// TIA Portal project "1_TIA" (V17)

(* hardware
DEVICE "S7-1200 station_1"  S7-1200 Station
   slot 0: "Rack_0"  S7-1200 Rack  Rack  V1.0
   slot 1: "STATION_1"  CPU 1215C DC/DC/DC  6ES7 215-1AG40-0XB0  V4.4
DEVICE "S7-1200 station_2"  S7-1200 Station
   slot 0: "Rack_0"  S7-1200 Rack  Rack  V1.0
   slot 1: "STATION_2"  CPU 1215C DC/DC/DC  6ES7 215-1AG40-0XB0  V4.4
*)

// ===== PLC "STATION_1"  CPU 1215C DC/DC/DC =====

VAR_GLOBAL   // PLC tag table "Default tag table"
   "Clock_Byte" AT %MB0 : Byte;
   "Clock_10Hz" AT %M0.0 : Bool;
   "Clock_5Hz" AT %M0.1 : Bool;
   "Clock_2.5Hz" AT %M0.2 : Bool;
   "Clock_2Hz" AT %M0.3 : Bool;
   "Clock_1.25Hz" AT %M0.4 : Bool;
   "Clock_1Hz" AT %M0.5 : Bool;
   "Clock_0.625Hz" AT %M0.6 : Bool;
   "Clock_0.5Hz" AT %M0.7 : Bool;
   "System_Byte" AT %MB1 : Byte;
   "FirstScan" AT %M1.0 : Bool;
   "DiagStatusUpdate" AT %M1.1 : Bool;
   "AlwaysTRUE" AT %M1.2 : Bool;
   "AlwaysFALSE" AT %M1.3 : Bool;
   "XUNG_PTRIG_1" AT %M10.0 : Bool;
   "XUNG_PTRIG_2" AT %M10.1 : Bool;
   "XUNG_PTRIG_3" AT %M10.2 : Bool;
   "XUNG_PTRIG_4" AT %M10.3 : Bool;
   "XUNG_PTRIG_5" AT %M10.4 : Bool;
   "XUNG_PTRIG_6" AT %M10.5 : Bool;
   "XUNG_PTRIG_7" AT %M10.6 : Bool;
   "XUNG_PTRIG_8" AT %M10.7 : Bool;
END_VAR

VAR_GLOBAL   // PLC tag table "Input"
   "Fault_Valve_1" AT %I0.0 : Bool;   // Bit báo lỗi van 1
   "Fault_Valve_2" AT %I0.1 : Bool;   // Bit báo lỗi van 2
   "Fault_Valve_3" AT %I0.2 : Bool;   // Bit báo lỗi van 3
   "FAULT_DC_TRON" AT %I0.3 : Bool;   // Bit báo lỗi động cơ trộn
   "Auto" AT %I0.5 : Bool;   // Chế độ Auto
   "Manual" AT %I0.6 : Bool;   // Chế độ Manual
   "FAULT_DC_EXPORT" AT %I0.4 : Bool;   // Bit baso lỗi máy đóng gói
   "ON" AT %I0.7 : Bool;   // Bật Hệ thống
   "OFF" AT %I1.0 : Bool;   // Tắt hệ thống
END_VAR

VAR_GLOBAL   // PLC tag table "Output"
   "Q_VALVE_1" AT %Q0.0 : Bool;   // Đầu ra van 1
   "Q_VALVE_2" AT %Q0.1 : Bool;   // Đầu ra van 2
   "Q_VALVE_3" AT %Q0.2 : Bool;   // Đầu ra van 3
   "Q_DC_TRON" AT %Q0.3 : Bool;   // Đầu ra động cơ trộn
   "Q_Lamp_Auto" AT %Q0.5 : Bool;
   "Q_Lamp_Manu" AT %Q0.6 : Bool;
   "Q_DC_Export" AT %Q0.4 : Bool;   // Đầu ra máy đóng gói
   "Q_System" AT %Q0.7 : Bool;
END_VAR

VAR_GLOBAL   // PLC tag table "simulation"
   "Simu_Fault_Valve_1" AT %M20.0 : Bool;
   "Simu_Fault_Valve_2" AT %M20.1 : Bool;
   "Simu_Fault_Valve_3" AT %M20.2 : Bool;
   "Simu_Fault_DC_TRON" AT %M20.3 : Bool;
   "Simu_Fault_DC_EXPORT" AT %M20.4 : Bool;
END_VAR

DATA_BLOCK "DB_Webserver"   // DB1
{ S7_Optimized_Access := 'FALSE' }
VERSION : 0.1
   VAR
      btt_Auto : Bool;   // Nút nhấn chế độ tự động
      btt_Manu : Bool;   // Nút nhấn chế độ bằng tay
      btt_Auto_Confirm : Bool;   // Nút nhấn xác nhận
      btt_V1_Open : Bool;   // Nút nhấn chế độ bằng tay mở van 1
      btt_V1_Close : Bool;   // Nút nhấn chế độ bằng tay đóng van 1
      btt_V2_Open : Bool;   // Nút nhấn chế độ bằng tay mở van 2
      btt_V2_Close : Bool;   // Nút nhấn chế độ bằng tay đóng van 2
      btt_V3_Open : Bool;   // Nút nhấn chế độ bằng tay mở van 3
      btt_V3_Close : Bool;   // Nút nhấn chế độ bằng tay đóng van 3
      btt_DC_Tron_Run : Bool;   // Nút nhấn chế độ bằng tay chạy ĐC trộn
      btt_DC_Tron_Stop : Bool;   // Nút nhấn chế độ bằng tay dừng ĐC trộn
      btt_DC_Export_Run : Bool;   // Nút nhấn chế độ bằng tay chạy máy đóng gói
      btt_DC_Export_Stop : Bool;   // Nút nhấn chế độ bằng tay đóng máy đóng gói
      CB_Can : Bool;   // Cảm biến cạn bồn trộn
      Q_Lamp_Auto : Bool;   // Đèn chế độ tự động
      Q_Lamp_Manu : Bool;   // Đèn chế độ bằng tay
      status_Valve_1 : Byte;   // Trạng thái van 1 (0 = Đang đóng, 1 = Đang mở, 2 = Đang lỗi)
      status_Valve_2 : Byte;   // Trạng thái van 2 (0 = Đang đóng, 1 = Đang mở, 2 = Đang lỗi)
      status_Valve_3 : Byte;   // Trạng thái van 3 (0 = Đang đóng, 1 = Đang mở, 2 = Đang lỗi)
      status_DC_Tron : Byte;   // Trạng thái ĐC trộn (0 = Đang đóng, 1 = Đang mở, 2 = Đang lỗi)
      status_DC_Export : Byte;   // Trạng thái Máy đóng gói (0 = Đang đóng, 1 = Đang mở, 2 = Đang lỗi)
      Setting_Time_Tron : Int := 10;   // Cài đặt thời gian trộn
      Act_Time_Tron : Int;   // Giá trị thực tế thời gian trộn
      Setting_Weight_1 : Real := 12.25;   // Cài đặt trọng lượng liệu 1
      Setting_Weight_2 : Real := 20.45;   // Cài đặt trọng lượng liệu 2
      Setting_Weight_3 : Real := 10.12;   // Cài đặt trọng lượng liệu 3
      Act_Weight_1 : Real;   // Giá trị thực tế trọng lượng liệu 1
      Act_Weight_2 : Real;   // Giá trị thực tế trọng lượng liệu 2
      Act_Weight_3 : Real;   // Giá trị thực tế trọng lượng liệu 3
      sql_insert_Trigger : Bool;   // Bit lưu giá trị lên SQL
      sql_insert_On : Bool;
      sql_insert_Off : Bool;
      sql_insert_Temp : Bool;
      sql_delete_Trigger : Bool;   // Bit xóa dữ liệu SQL
      sql_OrderID : String := 'Product 0';   // ID đơn hàng cần trộn
      sql_Weight1_Setting : Real;
      sql_Weight2_Setting : Real;
      sql_Weight3_Setting : Real;
      sql_Weight1_Actual : Real;
      sql_Weight2_Actual : Real;
      sql_Weight3_Actual : Real;
      sql_Time_Tron_Setting : Int;
      sql_Time_Tron_Actual : Int;
      on_System : Bool;
      off_System : Bool;
   END_VAR
BEGIN
END_DATA_BLOCK

DATA_BLOCK "Data"   // DB2
{ S7_Optimized_Access := 'TRUE' }
VERSION : 0.1
   VAR
      act_Step_1 : Bool;   // Giá trị thực tế bước 1
      act_Step_2 : Bool;   // Giá trị thực tế bước 2
      act_Step_3 : Bool;   // Giá trị thực tế bước 3
      act_done_valve_1 : Bool;   // Bit báo đã xả xong nguyên liệu 1
      act_done_valve_2 : Bool;   // Bit báo đã xả xong nguyên liệu 2
      act_done_valve_3 : Bool;   // Bit báo đã xả xong nguyên liệu 3
   END_VAR
BEGIN
END_DATA_BLOCK

DATA_BLOCK "DB_Alarm"   // DB4
{ S7_Optimized_Access := 'FALSE' }
VERSION : 0.1
   VAR
      Alarm_M1 : Bool;
      Alarm_M2 : Bool;
      Alarm_M3 : Bool;
      Alarm_Mix : Bool;
      Alarm_Export : Bool;
   END_VAR
BEGIN
END_DATA_BLOCK

// folder: System blocks/Program resources

DATA_BLOCK "TIMER_SIMU"   // DB3
{ S7_Optimized_Access := 'TRUE' }
AUTHOR : Simatic
FAMILY : IEC
NAME : IEC_TMR
VERSION : 1.0
// stored: InstanceOfName IEC_TIMER
"IEC_TIMER"
BEGIN
END_DATA_BLOCK

DATA_BLOCK "TImer_SQL_Delete"   // DB5
{ S7_Optimized_Access := 'TRUE' }
AUTHOR : Simatic
FAMILY : IEC
NAME : IEC_TMR
VERSION : 1.0
// stored: InstanceOfName IEC_TIMER
"IEC_TIMER"
BEGIN
END_DATA_BLOCK

DATA_BLOCK "sql_insert_on"   // DB6
{ S7_Optimized_Access := 'TRUE' }
AUTHOR : Simatic
FAMILY : IEC
NAME : IEC_TMR
VERSION : 1.0
// stored: InstanceOfName IEC_TIMER
"IEC_TIMER"
BEGIN
END_DATA_BLOCK

// folder: (top level)

FUNCTION "FC_MANUAL_MODE" : Void   // FC1, LAD
{ S7_Optimized_Access := 'TRUE' }
VERSION : 0.1
   VAR_TEMP   // added for the SCL form of the ladder/FBD networks
      _w1 : Bool;
      _w2 : Bool;
      _w3 : Bool;
      _w4 : Bool;
      _w5 : Bool;
      _w6 : Bool;
   END_VAR
BEGIN

REGION Network 1: Đầu ra động cơ trộn
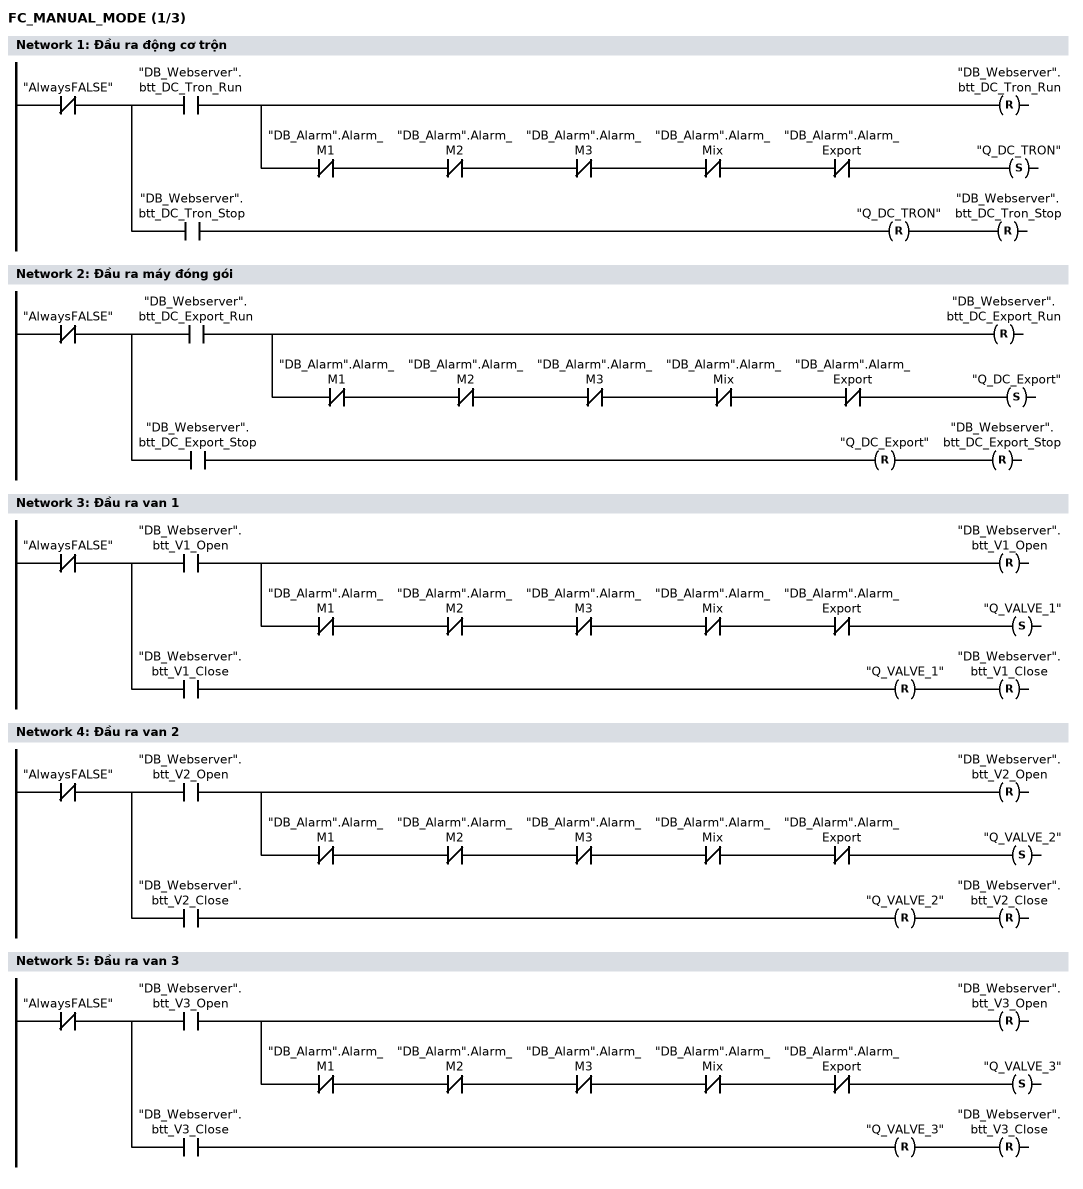
   RUNG wire#powerrail
      I_Contact( "AlwaysFALSE" )
      wire#w1
      Contact( "DB_Webserver".btt_DC_Tron_Run )
      wire#w2
      R_Coil( "DB_Webserver".btt_DC_Tron_Run )
   END_RUNG
   RUNG wire#w2
      I_Contact( "DB_Alarm".Alarm_M1 )
      I_Contact( "DB_Alarm".Alarm_M2 )
      I_Contact( "DB_Alarm".Alarm_M3 )
      I_Contact( "DB_Alarm".Alarm_Mix )
      I_Contact( "DB_Alarm".Alarm_Export )
      S_Coil( "Q_DC_TRON" )
   END_RUNG
   RUNG wire#w1
      Contact( "DB_Webserver".btt_DC_Tron_Stop )
      R_Coil( "Q_DC_TRON" )
      R_Coil( "DB_Webserver".btt_DC_Tron_Stop )
   END_RUNG
   // the same network as SCL:
   #_w1 := NOT "AlwaysFALSE" AND "DB_Webserver".btt_DC_Tron_Run;
   IF #_w1 THEN "DB_Webserver".btt_DC_Tron_Run := FALSE; END_IF;
   IF #_w1 AND NOT "DB_Alarm".Alarm_M1 AND NOT "DB_Alarm".Alarm_M2 AND NOT "DB_Alarm".Alarm_M3 AND NOT "DB_Alarm".Alarm_Mix AND NOT "DB_Alarm".Alarm_Export THEN
       "Q_DC_TRON" := TRUE;
   END_IF;
   IF NOT "AlwaysFALSE" AND "DB_Webserver".btt_DC_Tron_Stop THEN
       "Q_DC_TRON" := FALSE;
       "DB_Webserver".btt_DC_Tron_Stop := FALSE;
   END_IF;
END_REGION

REGION Network 2: Đầu ra máy đóng gói
   RUNG wire#powerrail
      I_Contact( "AlwaysFALSE" )
      wire#w1
      Contact( "DB_Webserver".btt_DC_Export_Run )
      wire#w2
      R_Coil( "DB_Webserver".btt_DC_Export_Run )
   END_RUNG
   RUNG wire#w2
      I_Contact( "DB_Alarm".Alarm_M1 )
      I_Contact( "DB_Alarm".Alarm_M2 )
      I_Contact( "DB_Alarm".Alarm_M3 )
      I_Contact( "DB_Alarm".Alarm_Mix )
      I_Contact( "DB_Alarm".Alarm_Export )
      S_Coil( "Q_DC_Export" )
   END_RUNG
   RUNG wire#w1
      Contact( "DB_Webserver".btt_DC_Export_Stop )
      R_Coil( "Q_DC_Export" )
      R_Coil( "DB_Webserver".btt_DC_Export_Stop )
   END_RUNG
   // the same network as SCL:
   #_w1 := NOT "AlwaysFALSE" AND "DB_Webserver".btt_DC_Export_Run;
   IF #_w1 THEN "DB_Webserver".btt_DC_Export_Run := FALSE; END_IF;
   IF #_w1 AND NOT "DB_Alarm".Alarm_M1 AND NOT "DB_Alarm".Alarm_M2 AND NOT "DB_Alarm".Alarm_M3 AND NOT "DB_Alarm".Alarm_Mix AND NOT "DB_Alarm".Alarm_Export THEN
       "Q_DC_Export" := TRUE;
   END_IF;
   IF NOT "AlwaysFALSE" AND "DB_Webserver".btt_DC_Export_Stop THEN
       "Q_DC_Export" := FALSE;
       "DB_Webserver".btt_DC_Export_Stop := FALSE;
   END_IF;
END_REGION

REGION Network 3: Đầu ra van 1
   RUNG wire#powerrail
      I_Contact( "AlwaysFALSE" )
      wire#w1
      Contact( "DB_Webserver".btt_V1_Open )
      wire#w2
      R_Coil( "DB_Webserver".btt_V1_Open )
   END_RUNG
   RUNG wire#w2
      I_Contact( "DB_Alarm".Alarm_M1 )
      I_Contact( "DB_Alarm".Alarm_M2 )
      I_Contact( "DB_Alarm".Alarm_M3 )
      I_Contact( "DB_Alarm".Alarm_Mix )
      I_Contact( "DB_Alarm".Alarm_Export )
      S_Coil( "Q_VALVE_1" )
   END_RUNG
   RUNG wire#w1
      Contact( "DB_Webserver".btt_V1_Close )
      R_Coil( "Q_VALVE_1" )
      R_Coil( "DB_Webserver".btt_V1_Close )
   END_RUNG
   // the same network as SCL:
   #_w1 := NOT "AlwaysFALSE" AND "DB_Webserver".btt_V1_Open;
   IF #_w1 THEN "DB_Webserver".btt_V1_Open := FALSE; END_IF;
   IF #_w1 AND NOT "DB_Alarm".Alarm_M1 AND NOT "DB_Alarm".Alarm_M2 AND NOT "DB_Alarm".Alarm_M3 AND NOT "DB_Alarm".Alarm_Mix AND NOT "DB_Alarm".Alarm_Export THEN
       "Q_VALVE_1" := TRUE;
   END_IF;
   IF NOT "AlwaysFALSE" AND "DB_Webserver".btt_V1_Close THEN
       "Q_VALVE_1" := FALSE;
       "DB_Webserver".btt_V1_Close := FALSE;
   END_IF;
END_REGION

REGION Network 4: Đầu ra van 2
   RUNG wire#powerrail
      I_Contact( "AlwaysFALSE" )
      wire#w1
      Contact( "DB_Webserver".btt_V2_Open )
      wire#w2
      R_Coil( "DB_Webserver".btt_V2_Open )
   END_RUNG
   RUNG wire#w2
      I_Contact( "DB_Alarm".Alarm_M1 )
      I_Contact( "DB_Alarm".Alarm_M2 )
      I_Contact( "DB_Alarm".Alarm_M3 )
      I_Contact( "DB_Alarm".Alarm_Mix )
      I_Contact( "DB_Alarm".Alarm_Export )
      S_Coil( "Q_VALVE_2" )
   END_RUNG
   RUNG wire#w1
      Contact( "DB_Webserver".btt_V2_Close )
      R_Coil( "Q_VALVE_2" )
      R_Coil( "DB_Webserver".btt_V2_Close )
   END_RUNG
   // the same network as SCL:
   #_w1 := NOT "AlwaysFALSE" AND "DB_Webserver".btt_V2_Open;
   IF #_w1 THEN "DB_Webserver".btt_V2_Open := FALSE; END_IF;
   IF #_w1 AND NOT "DB_Alarm".Alarm_M1 AND NOT "DB_Alarm".Alarm_M2 AND NOT "DB_Alarm".Alarm_M3 AND NOT "DB_Alarm".Alarm_Mix AND NOT "DB_Alarm".Alarm_Export THEN
       "Q_VALVE_2" := TRUE;
   END_IF;
   IF NOT "AlwaysFALSE" AND "DB_Webserver".btt_V2_Close THEN
       "Q_VALVE_2" := FALSE;
       "DB_Webserver".btt_V2_Close := FALSE;
   END_IF;
END_REGION

REGION Network 5: Đầu ra van 3
   RUNG wire#powerrail
      I_Contact( "AlwaysFALSE" )
      wire#w1
      Contact( "DB_Webserver".btt_V3_Open )
      wire#w2
      R_Coil( "DB_Webserver".btt_V3_Open )
   END_RUNG
   RUNG wire#w2
      I_Contact( "DB_Alarm".Alarm_M1 )
      I_Contact( "DB_Alarm".Alarm_M2 )
      I_Contact( "DB_Alarm".Alarm_M3 )
      I_Contact( "DB_Alarm".Alarm_Mix )
      I_Contact( "DB_Alarm".Alarm_Export )
      S_Coil( "Q_VALVE_3" )
   END_RUNG
   RUNG wire#w1
      Contact( "DB_Webserver".btt_V3_Close )
      R_Coil( "Q_VALVE_3" )
      R_Coil( "DB_Webserver".btt_V3_Close )
   END_RUNG
   // the same network as SCL:
   #_w1 := NOT "AlwaysFALSE" AND "DB_Webserver".btt_V3_Open;
   IF #_w1 THEN "DB_Webserver".btt_V3_Open := FALSE; END_IF;
   IF #_w1 AND NOT "DB_Alarm".Alarm_M1 AND NOT "DB_Alarm".Alarm_M2 AND NOT "DB_Alarm".Alarm_M3 AND NOT "DB_Alarm".Alarm_Mix AND NOT "DB_Alarm".Alarm_Export THEN
       "Q_VALVE_3" := TRUE;
   END_IF;
   IF NOT "AlwaysFALSE" AND "DB_Webserver".btt_V3_Close THEN
       "Q_VALVE_3" := FALSE;
       "DB_Webserver".btt_V3_Close := FALSE;
   END_IF;
END_REGION

REGION Network 6: mô phỏng tăng trọng lượng
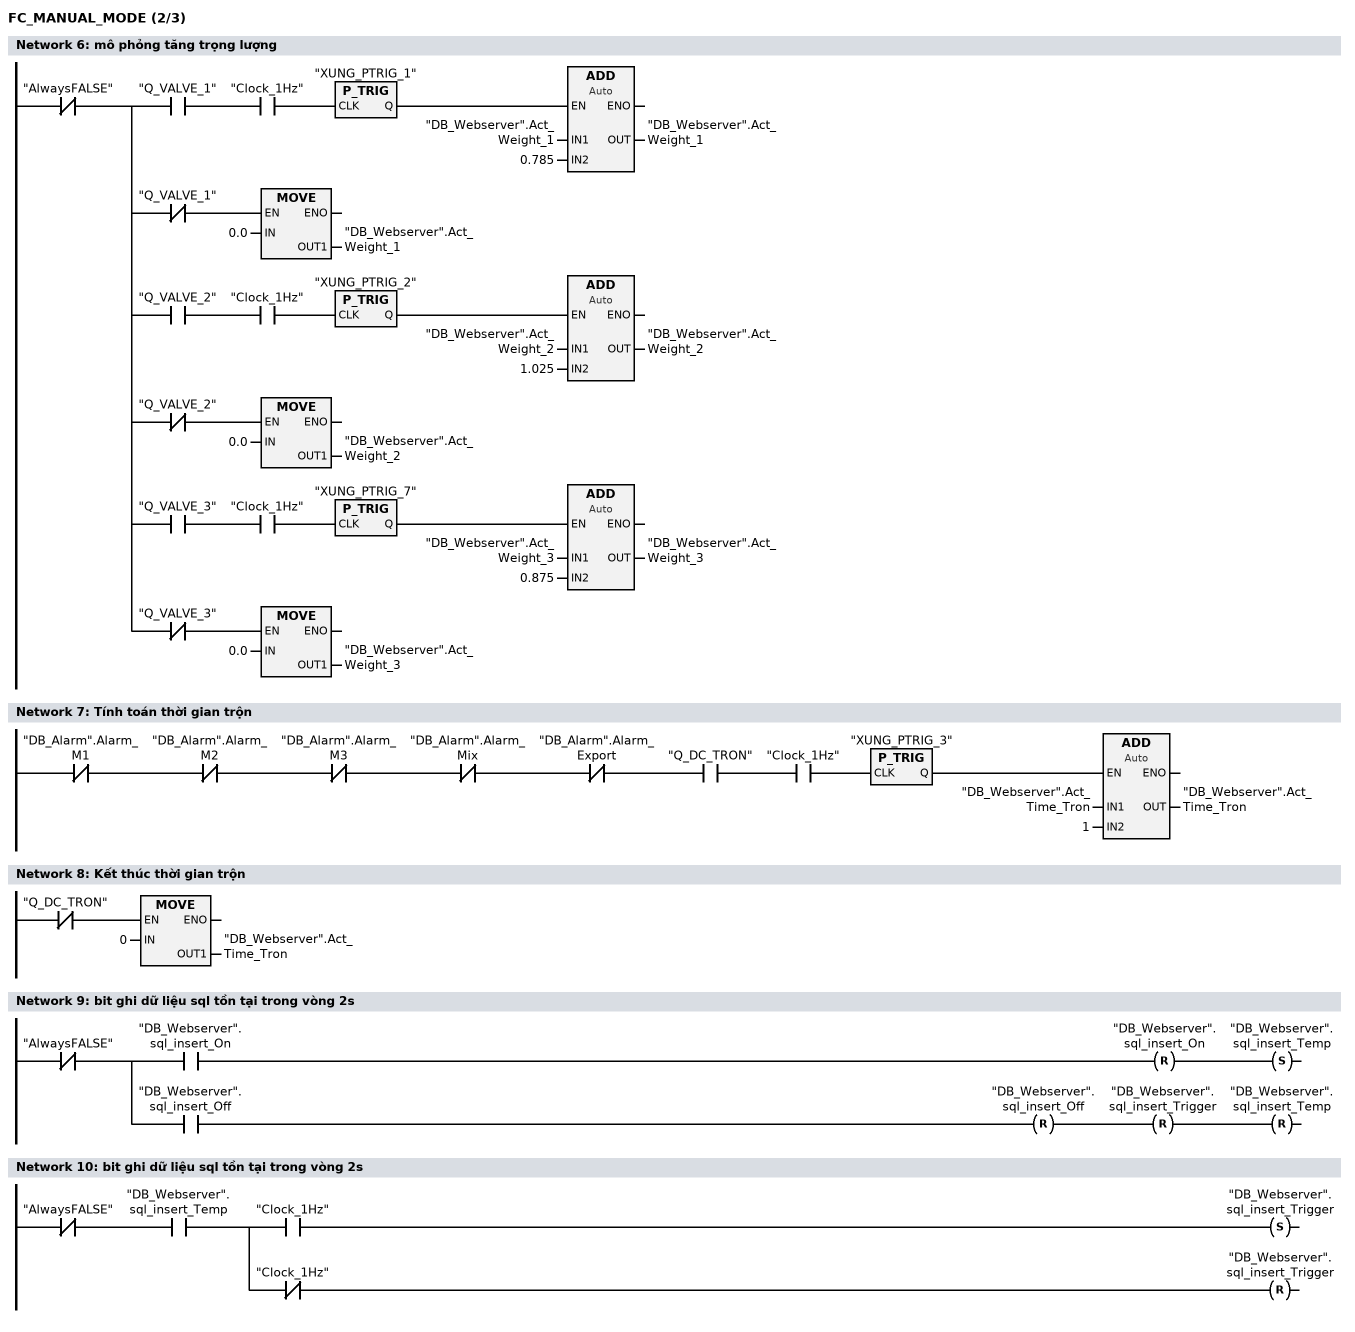
   RUNG wire#powerrail
      I_Contact( "AlwaysFALSE" )
      wire#w1
      Contact( "Q_VALVE_1" )
      Contact( "Clock_1Hz" )
      P_Trig( "XUNG_PTRIG_1" )
      Add(in1 := "DB_Webserver".Act_Weight_1, in2 := 0.785, out => "DB_Webserver".Act_Weight_1)
   END_RUNG
   RUNG wire#w1
      I_Contact( "Q_VALVE_1" )
      Move(in := 0.0, out1 => "DB_Webserver".Act_Weight_1)
   END_RUNG
   RUNG wire#w1
      Contact( "Q_VALVE_2" )
      Contact( "Clock_1Hz" )
      P_Trig( "XUNG_PTRIG_2" )
      Add(in1 := "DB_Webserver".Act_Weight_2, in2 := 1.025, out => "DB_Webserver".Act_Weight_2)
   END_RUNG
   RUNG wire#w1
      I_Contact( "Q_VALVE_2" )
      Move(in := 0.0, out1 => "DB_Webserver".Act_Weight_2)
   END_RUNG
   RUNG wire#w1
      Contact( "Q_VALVE_3" )
      Contact( "Clock_1Hz" )
      P_Trig( "XUNG_PTRIG_7" )
      Add(in1 := "DB_Webserver".Act_Weight_3, in2 := 0.875, out => "DB_Webserver".Act_Weight_3)
   END_RUNG
   RUNG wire#w1
      I_Contact( "Q_VALVE_3" )
      Move(in := 0.0, out1 => "DB_Webserver".Act_Weight_3)
   END_RUNG
   // the same network as SCL:
   #_w1 := NOT "AlwaysFALSE" AND "Q_VALVE_1" AND "Clock_1Hz";
   #_w2 := #_w1 AND NOT "XUNG_PTRIG_1";   // rising edge
   "XUNG_PTRIG_1" := #_w1;
   IF #_w2 THEN "DB_Webserver".Act_Weight_1 := "DB_Webserver".Act_Weight_1 + 0.785; END_IF;
   IF NOT "AlwaysFALSE" AND NOT "Q_VALVE_1" THEN "DB_Webserver".Act_Weight_1 := 0.0; END_IF;
   #_w3 := NOT "AlwaysFALSE" AND "Q_VALVE_2" AND "Clock_1Hz";
   #_w4 := #_w3 AND NOT "XUNG_PTRIG_2";   // rising edge
   "XUNG_PTRIG_2" := #_w3;
   IF #_w4 THEN "DB_Webserver".Act_Weight_2 := "DB_Webserver".Act_Weight_2 + 1.025; END_IF;
   IF NOT "AlwaysFALSE" AND NOT "Q_VALVE_2" THEN "DB_Webserver".Act_Weight_2 := 0.0; END_IF;
   #_w5 := NOT "AlwaysFALSE" AND "Q_VALVE_3" AND "Clock_1Hz";
   #_w6 := #_w5 AND NOT "XUNG_PTRIG_7";   // rising edge
   "XUNG_PTRIG_7" := #_w5;
   IF #_w6 THEN "DB_Webserver".Act_Weight_3 := "DB_Webserver".Act_Weight_3 + 0.875; END_IF;
   IF NOT "AlwaysFALSE" AND NOT "Q_VALVE_3" THEN "DB_Webserver".Act_Weight_3 := 0.0; END_IF;
END_REGION

REGION Network 7: Tính toán thời gian trộn
   RUNG wire#powerrail
      I_Contact( "DB_Alarm".Alarm_M1 )
      I_Contact( "DB_Alarm".Alarm_M2 )
      I_Contact( "DB_Alarm".Alarm_M3 )
      I_Contact( "DB_Alarm".Alarm_Mix )
      I_Contact( "DB_Alarm".Alarm_Export )
      Contact( "Q_DC_TRON" )
      Contact( "Clock_1Hz" )
      P_Trig( "XUNG_PTRIG_3" )
      Add(in1 := "DB_Webserver".Act_Time_Tron, in2 := 1, out => "DB_Webserver".Act_Time_Tron)
   END_RUNG
   // the same network as SCL:
   #_w1 := NOT "DB_Alarm".Alarm_M1 AND NOT "DB_Alarm".Alarm_M2 AND NOT "DB_Alarm".Alarm_M3 AND NOT "DB_Alarm".Alarm_Mix AND NOT "DB_Alarm".Alarm_Export AND "Q_DC_TRON" AND "Clock_1Hz";
   #_w2 := #_w1 AND NOT "XUNG_PTRIG_3";   // rising edge
   "XUNG_PTRIG_3" := #_w1;
   IF #_w2 THEN "DB_Webserver".Act_Time_Tron := "DB_Webserver".Act_Time_Tron + 1; END_IF;
END_REGION

REGION Network 8: Kết thúc thời gian trộn
   RUNG wire#powerrail
      I_Contact( "Q_DC_TRON" )
      Move(in := 0, out1 => "DB_Webserver".Act_Time_Tron)
   END_RUNG
   // the same network as SCL:
   IF NOT "Q_DC_TRON" THEN "DB_Webserver".Act_Time_Tron := 0; END_IF;
END_REGION

REGION Network 9: bit ghi dữ liệu sql tồn tại trong vòng 2s
   RUNG wire#powerrail
      I_Contact( "AlwaysFALSE" )
      wire#w1
      Contact( "DB_Webserver".sql_insert_On )
      R_Coil( "DB_Webserver".sql_insert_On )
      S_Coil( "DB_Webserver".sql_insert_Temp )
   END_RUNG
   RUNG wire#w1
      Contact( "DB_Webserver".sql_insert_Off )
      R_Coil( "DB_Webserver".sql_insert_Off )
      R_Coil( "DB_Webserver".sql_insert_Trigger )
      R_Coil( "DB_Webserver".sql_insert_Temp )
   END_RUNG
   // the same network as SCL:
   #_w1 := NOT "AlwaysFALSE" AND "DB_Webserver".sql_insert_On;
   IF #_w1 THEN
       "DB_Webserver".sql_insert_On := FALSE;
       "DB_Webserver".sql_insert_Temp := TRUE;
   END_IF;
   #_w2 := NOT "AlwaysFALSE" AND "DB_Webserver".sql_insert_Off;
   IF #_w2 THEN
       "DB_Webserver".sql_insert_Off := FALSE;
       "DB_Webserver".sql_insert_Trigger := FALSE;
       "DB_Webserver".sql_insert_Temp := FALSE;
   END_IF;
END_REGION

REGION Network 10: bit ghi dữ liệu sql tồn tại trong vòng 2s
   RUNG wire#powerrail
      I_Contact( "AlwaysFALSE" )
      Contact( "DB_Webserver".sql_insert_Temp )
      wire#w1
      Contact( "Clock_1Hz" )
      S_Coil( "DB_Webserver".sql_insert_Trigger )
   END_RUNG
   RUNG wire#w1
      I_Contact( "Clock_1Hz" )
      R_Coil( "DB_Webserver".sql_insert_Trigger )
   END_RUNG
   // the same network as SCL:
   #_w1 := NOT "AlwaysFALSE" AND "DB_Webserver".sql_insert_Temp;
   IF #_w1 AND "Clock_1Hz" THEN "DB_Webserver".sql_insert_Trigger := TRUE; END_IF;
   IF #_w1 AND NOT "Clock_1Hz" THEN "DB_Webserver".sql_insert_Trigger := FALSE; END_IF;
END_REGION

REGION Network 11: bit ghi dữ liệu sql tồn tại trong vòng 2s
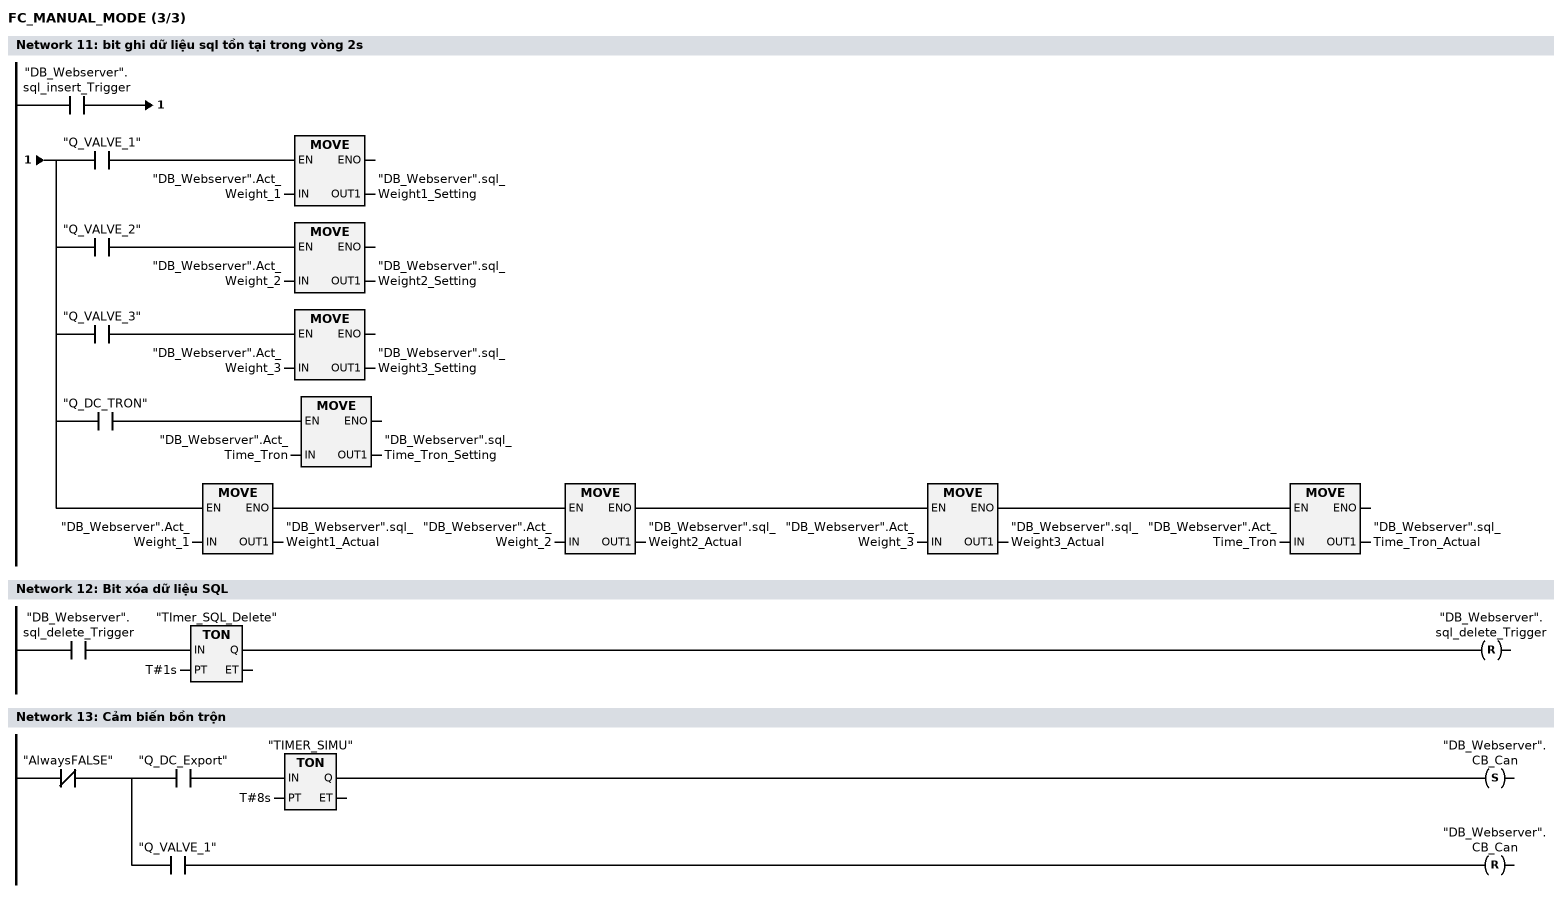
   RUNG wire#powerrail
      Contact( "DB_Webserver".sql_insert_Trigger )
      wire#w1
      Contact( "Q_VALVE_1" )
      Move(in := "DB_Webserver".Act_Weight_1, out1 => "DB_Webserver".sql_Weight1_Setting)
   END_RUNG
   RUNG wire#w1
      Contact( "Q_VALVE_2" )
      Move(in := "DB_Webserver".Act_Weight_2, out1 => "DB_Webserver".sql_Weight2_Setting)
   END_RUNG
   RUNG wire#w1
      Contact( "Q_VALVE_3" )
      Move(in := "DB_Webserver".Act_Weight_3, out1 => "DB_Webserver".sql_Weight3_Setting)
   END_RUNG
   RUNG wire#w1
      Contact( "Q_DC_TRON" )
      Move(in := "DB_Webserver".Act_Time_Tron, out1 => "DB_Webserver".sql_Time_Tron_Setting)
   END_RUNG
   RUNG wire#w1
      Move(in := "DB_Webserver".Act_Weight_1, out1 => "DB_Webserver".sql_Weight1_Actual)
      Move(in := "DB_Webserver".Act_Weight_2, out1 => "DB_Webserver".sql_Weight2_Actual)
      Move(in := "DB_Webserver".Act_Weight_3, out1 => "DB_Webserver".sql_Weight3_Actual)
      Move(in := "DB_Webserver".Act_Time_Tron, out1 => "DB_Webserver".sql_Time_Tron_Actual)
   END_RUNG
   // the same network as SCL:
   IF "DB_Webserver".sql_insert_Trigger AND "Q_VALVE_1" THEN
       "DB_Webserver".sql_Weight1_Setting := "DB_Webserver".Act_Weight_1;
   END_IF;
   IF "DB_Webserver".sql_insert_Trigger AND "Q_VALVE_2" THEN
       "DB_Webserver".sql_Weight2_Setting := "DB_Webserver".Act_Weight_2;
   END_IF;
   IF "DB_Webserver".sql_insert_Trigger AND "Q_VALVE_3" THEN
       "DB_Webserver".sql_Weight3_Setting := "DB_Webserver".Act_Weight_3;
   END_IF;
   IF "DB_Webserver".sql_insert_Trigger AND "Q_DC_TRON" THEN
       "DB_Webserver".sql_Time_Tron_Setting := "DB_Webserver".Act_Time_Tron;
   END_IF;
   IF "DB_Webserver".sql_insert_Trigger THEN
       "DB_Webserver".sql_Weight1_Actual := "DB_Webserver".Act_Weight_1;
       "DB_Webserver".sql_Weight2_Actual := "DB_Webserver".Act_Weight_2;
       "DB_Webserver".sql_Weight3_Actual := "DB_Webserver".Act_Weight_3;
       "DB_Webserver".sql_Time_Tron_Actual := "DB_Webserver".Act_Time_Tron;
   END_IF;
END_REGION

REGION Network 12: Bit xóa dữ liệu SQL
   "TImer_SQL_Delete".TON(IN := "DB_Webserver".sql_delete_Trigger, PT := T#1s);
   IF "TImer_SQL_Delete".Q THEN "DB_Webserver".sql_delete_Trigger := FALSE; END_IF;
END_REGION

REGION Network 13: Cảm biến bồn trộn
   "TIMER_SIMU".TON(IN := NOT "AlwaysFALSE" AND "Q_DC_Export", PT := T#8s);
   IF "TIMER_SIMU".Q THEN "DB_Webserver".CB_Can := TRUE; END_IF;
   IF NOT "AlwaysFALSE" AND "Q_VALVE_1" THEN "DB_Webserver".CB_Can := FALSE; END_IF;
END_REGION
END_FUNCTION

FUNCTION "FC_AUTO_MODE" : Void   // FC2, LAD
{ S7_Optimized_Access := 'TRUE' }
VERSION : 0.1
   VAR_TEMP   // added for the SCL form of the ladder/FBD networks
      _w1 : Bool;
      _w2 : Bool;
      _w3 : Bool;
      _w4 : Bool;
      _w5 : Bool;
      _w6 : Bool;
   END_VAR
BEGIN

REGION Network 1: mô phỏng tăng trọng lượng
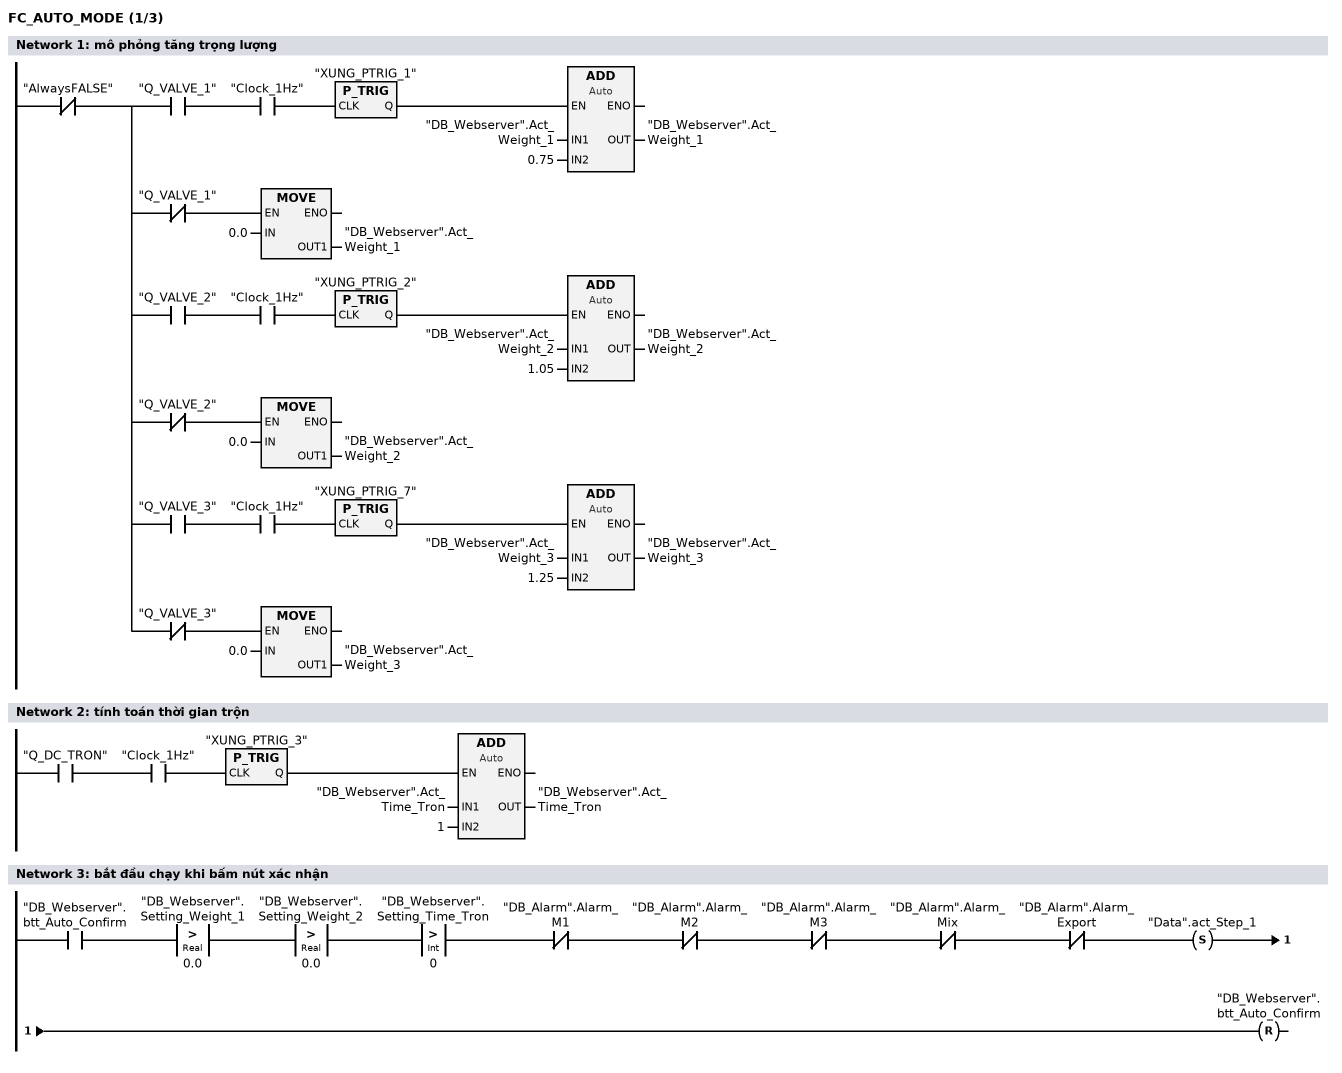
   RUNG wire#powerrail
      I_Contact( "AlwaysFALSE" )
      wire#w1
      Contact( "Q_VALVE_1" )
      Contact( "Clock_1Hz" )
      P_Trig( "XUNG_PTRIG_1" )
      Add(in1 := "DB_Webserver".Act_Weight_1, in2 := 0.75, out => "DB_Webserver".Act_Weight_1)
   END_RUNG
   RUNG wire#w1
      I_Contact( "Q_VALVE_1" )
      Move(in := 0.0, out1 => "DB_Webserver".Act_Weight_1)
   END_RUNG
   RUNG wire#w1
      Contact( "Q_VALVE_2" )
      Contact( "Clock_1Hz" )
      P_Trig( "XUNG_PTRIG_2" )
      Add(in1 := "DB_Webserver".Act_Weight_2, in2 := 1.05, out => "DB_Webserver".Act_Weight_2)
   END_RUNG
   RUNG wire#w1
      I_Contact( "Q_VALVE_2" )
      Move(in := 0.0, out1 => "DB_Webserver".Act_Weight_2)
   END_RUNG
   RUNG wire#w1
      Contact( "Q_VALVE_3" )
      Contact( "Clock_1Hz" )
      P_Trig( "XUNG_PTRIG_7" )
      Add(in1 := "DB_Webserver".Act_Weight_3, in2 := 1.25, out => "DB_Webserver".Act_Weight_3)
   END_RUNG
   RUNG wire#w1
      I_Contact( "Q_VALVE_3" )
      Move(in := 0.0, out1 => "DB_Webserver".Act_Weight_3)
   END_RUNG
   // the same network as SCL:
   #_w1 := NOT "AlwaysFALSE" AND "Q_VALVE_1" AND "Clock_1Hz";
   #_w2 := #_w1 AND NOT "XUNG_PTRIG_1";   // rising edge
   "XUNG_PTRIG_1" := #_w1;
   IF #_w2 THEN "DB_Webserver".Act_Weight_1 := "DB_Webserver".Act_Weight_1 + 0.75; END_IF;
   IF NOT "AlwaysFALSE" AND NOT "Q_VALVE_1" THEN "DB_Webserver".Act_Weight_1 := 0.0; END_IF;
   #_w3 := NOT "AlwaysFALSE" AND "Q_VALVE_2" AND "Clock_1Hz";
   #_w4 := #_w3 AND NOT "XUNG_PTRIG_2";   // rising edge
   "XUNG_PTRIG_2" := #_w3;
   IF #_w4 THEN "DB_Webserver".Act_Weight_2 := "DB_Webserver".Act_Weight_2 + 1.05; END_IF;
   IF NOT "AlwaysFALSE" AND NOT "Q_VALVE_2" THEN "DB_Webserver".Act_Weight_2 := 0.0; END_IF;
   #_w5 := NOT "AlwaysFALSE" AND "Q_VALVE_3" AND "Clock_1Hz";
   #_w6 := #_w5 AND NOT "XUNG_PTRIG_7";   // rising edge
   "XUNG_PTRIG_7" := #_w5;
   IF #_w6 THEN "DB_Webserver".Act_Weight_3 := "DB_Webserver".Act_Weight_3 + 1.25; END_IF;
   IF NOT "AlwaysFALSE" AND NOT "Q_VALVE_3" THEN "DB_Webserver".Act_Weight_3 := 0.0; END_IF;
END_REGION

REGION Network 2: tính toán thời gian trộn
   RUNG wire#powerrail
      Contact( "Q_DC_TRON" )
      Contact( "Clock_1Hz" )
      P_Trig( "XUNG_PTRIG_3" )
      Add(in1 := "DB_Webserver".Act_Time_Tron, in2 := 1, out => "DB_Webserver".Act_Time_Tron)
   END_RUNG
   // the same network as SCL:
   #_w1 := "Q_DC_TRON" AND "Clock_1Hz";
   #_w2 := #_w1 AND NOT "XUNG_PTRIG_3";   // rising edge
   "XUNG_PTRIG_3" := #_w1;
   IF #_w2 THEN "DB_Webserver".Act_Time_Tron := "DB_Webserver".Act_Time_Tron + 1; END_IF;
END_REGION

REGION Network 3: bắt đầu chạy khi bấm nút xác nhận
   RUNG wire#powerrail
      Contact( "DB_Webserver".btt_Auto_Confirm )
      { S7_Templates := "SrcType := Real" } GT_Contact(in1 := "DB_Webserver".Setting_Weight_1, in2 := 0.0)
      { S7_Templates := "SrcType := Real" } GT_Contact(in1 := "DB_Webserver".Setting_Weight_2, in2 := 0.0)
      { S7_Templates := "SrcType := Int" } GT_Contact(in1 := "DB_Webserver".Setting_Time_Tron, in2 := 0)
      I_Contact( "DB_Alarm".Alarm_M1 )
      I_Contact( "DB_Alarm".Alarm_M2 )
      I_Contact( "DB_Alarm".Alarm_M3 )
      I_Contact( "DB_Alarm".Alarm_Mix )
      I_Contact( "DB_Alarm".Alarm_Export )
      S_Coil( "Data".act_Step_1 )
      R_Coil( "DB_Webserver".btt_Auto_Confirm )
   END_RUNG
   // the same network as SCL:
   IF "DB_Webserver".btt_Auto_Confirm AND ("DB_Webserver".Setting_Weight_1 > 0.0) AND ("DB_Webserver".Setting_Weight_2 > 0.0) AND ("DB_Webserver".Setting_Time_Tron > 0) AND NOT "DB_Alarm".Alarm_M1 AND NOT "DB_Alarm".Alarm_M2 AND NOT "DB_Alarm".Alarm_M3 AND NOT "DB_Alarm".Alarm_Mix AND NOT "DB_Alarm".Alarm_Export THEN
       "Data".act_Step_1 := TRUE;
       "DB_Webserver".btt_Auto_Confirm := FALSE;
   END_IF;
END_REGION

REGION Network 4: Giai đoạn 1
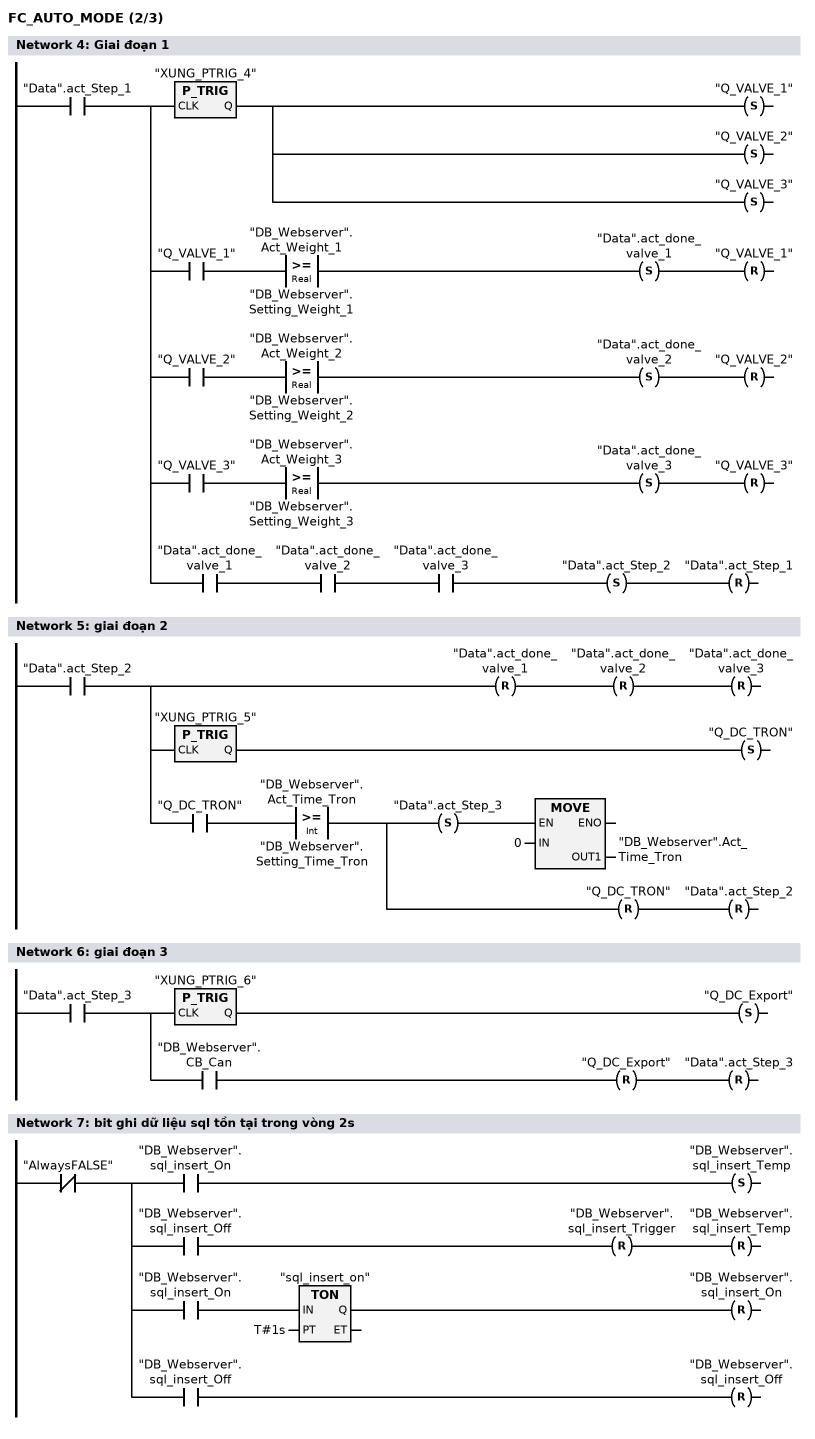
   RUNG wire#powerrail
      Contact( "Data".act_Step_1 )
      wire#w1
      P_Trig( "XUNG_PTRIG_4" )
      wire#w2
      S_Coil( "Q_VALVE_1" )
   END_RUNG
   RUNG wire#w2
      S_Coil( "Q_VALVE_2" )
   END_RUNG
   RUNG wire#w2
      S_Coil( "Q_VALVE_3" )
   END_RUNG
   RUNG wire#w1
      Contact( "Q_VALVE_1" )
      { S7_Templates := "SrcType := Real" } GE_Contact(in1 := "DB_Webserver".Act_Weight_1, in2 := "DB_Webserver".Setting_Weight_1)
      S_Coil( "Data".act_done_valve_1 )
      R_Coil( "Q_VALVE_1" )
   END_RUNG
   RUNG wire#w1
      Contact( "Q_VALVE_2" )
      { S7_Templates := "SrcType := Real" } GE_Contact(in1 := "DB_Webserver".Act_Weight_2, in2 := "DB_Webserver".Setting_Weight_2)
      S_Coil( "Data".act_done_valve_2 )
      R_Coil( "Q_VALVE_2" )
   END_RUNG
   RUNG wire#w1
      Contact( "Q_VALVE_3" )
      { S7_Templates := "SrcType := Real" } GE_Contact(in1 := "DB_Webserver".Act_Weight_3, in2 := "DB_Webserver".Setting_Weight_3)
      S_Coil( "Data".act_done_valve_3 )
      R_Coil( "Q_VALVE_3" )
   END_RUNG
   RUNG wire#w1
      Contact( "Data".act_done_valve_1 )
      Contact( "Data".act_done_valve_2 )
      Contact( "Data".act_done_valve_3 )
      S_Coil( "Data".act_Step_2 )
      R_Coil( "Data".act_Step_1 )
   END_RUNG
   // the same network as SCL:
   #_w1 := "Data".act_Step_1 AND NOT "XUNG_PTRIG_4";   // rising edge
   "XUNG_PTRIG_4" := "Data".act_Step_1;
   IF #_w1 THEN
       "Q_VALVE_1" := TRUE;
       "Q_VALVE_2" := TRUE;
       "Q_VALVE_3" := TRUE;
   END_IF;
   IF "Data".act_Step_1 AND "Q_VALVE_1" AND ("DB_Webserver".Act_Weight_1 >= "DB_Webserver".Setting_Weight_1) THEN
       "Data".act_done_valve_1 := TRUE;
       "Q_VALVE_1" := FALSE;
   END_IF;
   IF "Data".act_Step_1 AND "Q_VALVE_2" AND ("DB_Webserver".Act_Weight_2 >= "DB_Webserver".Setting_Weight_2) THEN
       "Data".act_done_valve_2 := TRUE;
       "Q_VALVE_2" := FALSE;
   END_IF;
   IF "Data".act_Step_1 AND "Q_VALVE_3" AND ("DB_Webserver".Act_Weight_3 >= "DB_Webserver".Setting_Weight_3) THEN
       "Data".act_done_valve_3 := TRUE;
       "Q_VALVE_3" := FALSE;
   END_IF;
   IF "Data".act_Step_1 AND "Data".act_done_valve_1 AND "Data".act_done_valve_2 AND "Data".act_done_valve_3 THEN
       "Data".act_Step_2 := TRUE;
       "Data".act_Step_1 := FALSE;
   END_IF;
END_REGION

REGION Network 5: giai đoạn 2
   RUNG wire#powerrail
      Contact( "Data".act_Step_2 )
      wire#w1
      R_Coil( "Data".act_done_valve_1 )
      R_Coil( "Data".act_done_valve_2 )
      R_Coil( "Data".act_done_valve_3 )
   END_RUNG
   RUNG wire#w1
      P_Trig( "XUNG_PTRIG_5" )
      S_Coil( "Q_DC_TRON" )
   END_RUNG
   RUNG wire#w1
      Contact( "Q_DC_TRON" )
      { S7_Templates := "SrcType := Int" } GE_Contact(in1 := "DB_Webserver".Act_Time_Tron, in2 := "DB_Webserver".Setting_Time_Tron)
      wire#w2
      S_Coil( "Data".act_Step_3 )
      Move(in := 0, out1 => "DB_Webserver".Act_Time_Tron)
   END_RUNG
   RUNG wire#w2
      R_Coil( "Q_DC_TRON" )
      R_Coil( "Data".act_Step_2 )
   END_RUNG
   // the same network as SCL:
   IF "Data".act_Step_2 THEN
       "Data".act_done_valve_1 := FALSE;
       "Data".act_done_valve_2 := FALSE;
       "Data".act_done_valve_3 := FALSE;
   END_IF;
   #_w1 := "Data".act_Step_2 AND NOT "XUNG_PTRIG_5";   // rising edge
   "XUNG_PTRIG_5" := "Data".act_Step_2;
   IF #_w1 THEN "Q_DC_TRON" := TRUE; END_IF;
   IF "Data".act_Step_2 AND "Q_DC_TRON" AND ("DB_Webserver".Act_Time_Tron >= "DB_Webserver".Setting_Time_Tron) THEN
       "Data".act_Step_3 := TRUE;
   END_IF;
   #_w2 := "Data".act_Step_2 AND "Q_DC_TRON" AND ("DB_Webserver".Act_Time_Tron >= "DB_Webserver".Setting_Time_Tron);
   IF #_w2 THEN
       "DB_Webserver".Act_Time_Tron := 0;
       "Q_DC_TRON" := FALSE;
       "Data".act_Step_2 := FALSE;
   END_IF;
END_REGION

REGION Network 6: giai đoạn 3
   RUNG wire#powerrail
      Contact( "Data".act_Step_3 )
      wire#w1
      P_Trig( "XUNG_PTRIG_6" )
      S_Coil( "Q_DC_Export" )
   END_RUNG
   RUNG wire#w1
      Contact( "DB_Webserver".CB_Can )
      R_Coil( "Q_DC_Export" )
      R_Coil( "Data".act_Step_3 )
   END_RUNG
   // the same network as SCL:
   #_w1 := "Data".act_Step_3 AND NOT "XUNG_PTRIG_6";   // rising edge
   "XUNG_PTRIG_6" := "Data".act_Step_3;
   IF #_w1 THEN "Q_DC_Export" := TRUE; END_IF;
   IF "Data".act_Step_3 AND "DB_Webserver".CB_Can THEN
       "Q_DC_Export" := FALSE;
       "Data".act_Step_3 := FALSE;
   END_IF;
END_REGION

REGION Network 7: bit ghi dữ liệu sql tồn tại trong vòng 2s
   IF NOT "AlwaysFALSE" AND "DB_Webserver".sql_insert_On THEN "DB_Webserver".sql_insert_Temp := TRUE; END_IF;
   IF NOT "AlwaysFALSE" AND "DB_Webserver".sql_insert_Off THEN
       "DB_Webserver".sql_insert_Trigger := FALSE;
       "DB_Webserver".sql_insert_Temp := FALSE;
   END_IF;
   "sql_insert_on".TON(IN := NOT "AlwaysFALSE" AND "DB_Webserver".sql_insert_On, PT := T#1s);
   IF "sql_insert_on".Q THEN "DB_Webserver".sql_insert_On := FALSE; END_IF;
   IF NOT "AlwaysFALSE" AND "DB_Webserver".sql_insert_Off THEN
       "DB_Webserver".sql_insert_Off := FALSE;
   END_IF;
END_REGION

REGION Network 8: bit ghi dữ liệu sql tồn tại trong vòng 2s
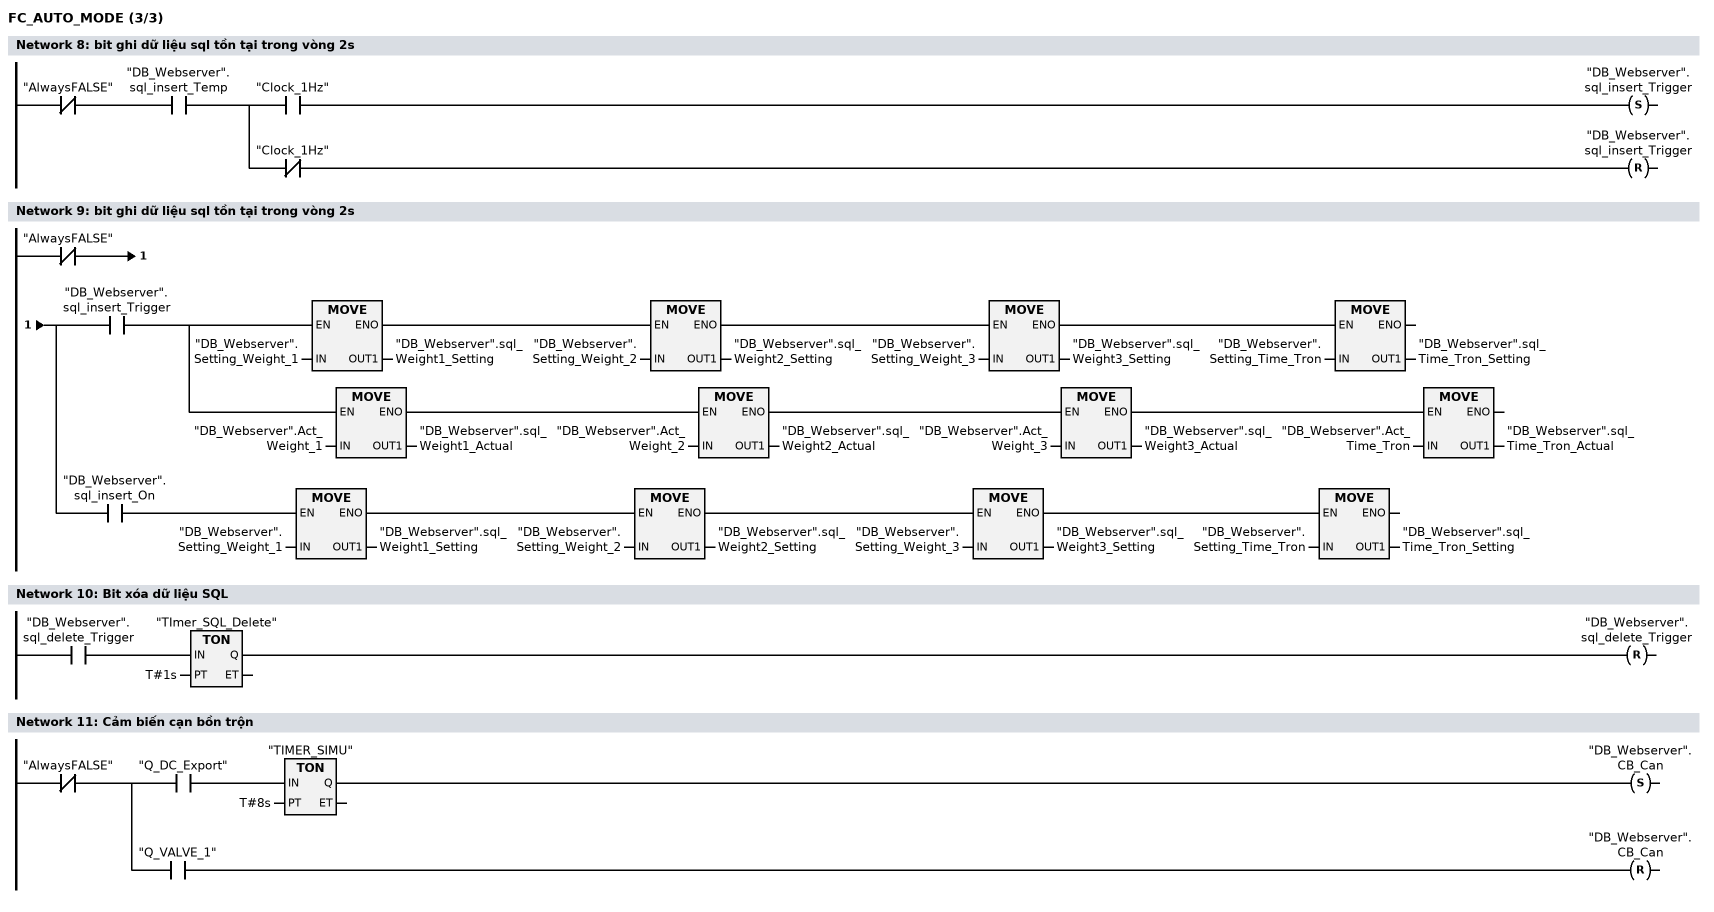
   RUNG wire#powerrail
      I_Contact( "AlwaysFALSE" )
      Contact( "DB_Webserver".sql_insert_Temp )
      wire#w1
      Contact( "Clock_1Hz" )
      S_Coil( "DB_Webserver".sql_insert_Trigger )
   END_RUNG
   RUNG wire#w1
      I_Contact( "Clock_1Hz" )
      R_Coil( "DB_Webserver".sql_insert_Trigger )
   END_RUNG
   // the same network as SCL:
   #_w1 := NOT "AlwaysFALSE" AND "DB_Webserver".sql_insert_Temp;
   IF #_w1 AND "Clock_1Hz" THEN "DB_Webserver".sql_insert_Trigger := TRUE; END_IF;
   IF #_w1 AND NOT "Clock_1Hz" THEN "DB_Webserver".sql_insert_Trigger := FALSE; END_IF;
END_REGION

REGION Network 9: bit ghi dữ liệu sql tồn tại trong vòng 2s
   RUNG wire#powerrail
      I_Contact( "AlwaysFALSE" )
      wire#w1
      Contact( "DB_Webserver".sql_insert_Trigger )
      wire#w2
      Move(in := "DB_Webserver".Setting_Weight_1, out1 => "DB_Webserver".sql_Weight1_Setting)
      Move(in := "DB_Webserver".Setting_Weight_2, out1 => "DB_Webserver".sql_Weight2_Setting)
      Move(in := "DB_Webserver".Setting_Weight_3, out1 => "DB_Webserver".sql_Weight3_Setting)
      Move(in := "DB_Webserver".Setting_Time_Tron, out1 => "DB_Webserver".sql_Time_Tron_Setting)
   END_RUNG
   RUNG wire#w2
      Move(in := "DB_Webserver".Act_Weight_1, out1 => "DB_Webserver".sql_Weight1_Actual)
      Move(in := "DB_Webserver".Act_Weight_2, out1 => "DB_Webserver".sql_Weight2_Actual)
      Move(in := "DB_Webserver".Act_Weight_3, out1 => "DB_Webserver".sql_Weight3_Actual)
      Move(in := "DB_Webserver".Act_Time_Tron, out1 => "DB_Webserver".sql_Time_Tron_Actual)
   END_RUNG
   RUNG wire#w1
      Contact( "DB_Webserver".sql_insert_On )
      Move(in := "DB_Webserver".Setting_Weight_1, out1 => "DB_Webserver".sql_Weight1_Setting)
      Move(in := "DB_Webserver".Setting_Weight_2, out1 => "DB_Webserver".sql_Weight2_Setting)
      Move(in := "DB_Webserver".Setting_Weight_3, out1 => "DB_Webserver".sql_Weight3_Setting)
      Move(in := "DB_Webserver".Setting_Time_Tron, out1 => "DB_Webserver".sql_Time_Tron_Setting)
   END_RUNG
   // the same network as SCL:
   IF NOT "AlwaysFALSE" AND "DB_Webserver".sql_insert_Trigger THEN
       "DB_Webserver".sql_Weight1_Setting := "DB_Webserver".Setting_Weight_1;
       "DB_Webserver".sql_Weight2_Setting := "DB_Webserver".Setting_Weight_2;
       "DB_Webserver".sql_Weight3_Setting := "DB_Webserver".Setting_Weight_3;
       "DB_Webserver".sql_Time_Tron_Setting := "DB_Webserver".Setting_Time_Tron;
       "DB_Webserver".sql_Weight1_Actual := "DB_Webserver".Act_Weight_1;
       "DB_Webserver".sql_Weight2_Actual := "DB_Webserver".Act_Weight_2;
       "DB_Webserver".sql_Weight3_Actual := "DB_Webserver".Act_Weight_3;
       "DB_Webserver".sql_Time_Tron_Actual := "DB_Webserver".Act_Time_Tron;
   END_IF;
   IF NOT "AlwaysFALSE" AND "DB_Webserver".sql_insert_On THEN
       "DB_Webserver".sql_Weight1_Setting := "DB_Webserver".Setting_Weight_1;
       "DB_Webserver".sql_Weight2_Setting := "DB_Webserver".Setting_Weight_2;
       "DB_Webserver".sql_Weight3_Setting := "DB_Webserver".Setting_Weight_3;
       "DB_Webserver".sql_Time_Tron_Setting := "DB_Webserver".Setting_Time_Tron;
   END_IF;
END_REGION

REGION Network 10: Bit xóa dữ liệu SQL
   "TImer_SQL_Delete".TON(IN := "DB_Webserver".sql_delete_Trigger, PT := T#1s);
   IF "TImer_SQL_Delete".Q THEN "DB_Webserver".sql_delete_Trigger := FALSE; END_IF;
END_REGION

REGION Network 11: Cảm biến cạn bồn trộn
   "TIMER_SIMU".TON(IN := NOT "AlwaysFALSE" AND "Q_DC_Export", PT := T#8s);
   IF "TIMER_SIMU".Q THEN "DB_Webserver".CB_Can := TRUE; END_IF;
   IF NOT "AlwaysFALSE" AND "Q_VALVE_1" THEN "DB_Webserver".CB_Can := FALSE; END_IF;
END_REGION
END_FUNCTION

FUNCTION "FC_EQUIPMENT_STATUS" : Void   // FC3, LAD
{ S7_Optimized_Access := 'TRUE' }
VERSION : 0.1
   VAR_TEMP   // added for the SCL form of the ladder/FBD networks
      _w1 : Bool;
   END_VAR
BEGIN

REGION Network 1: hiển thị trạng thái đèn
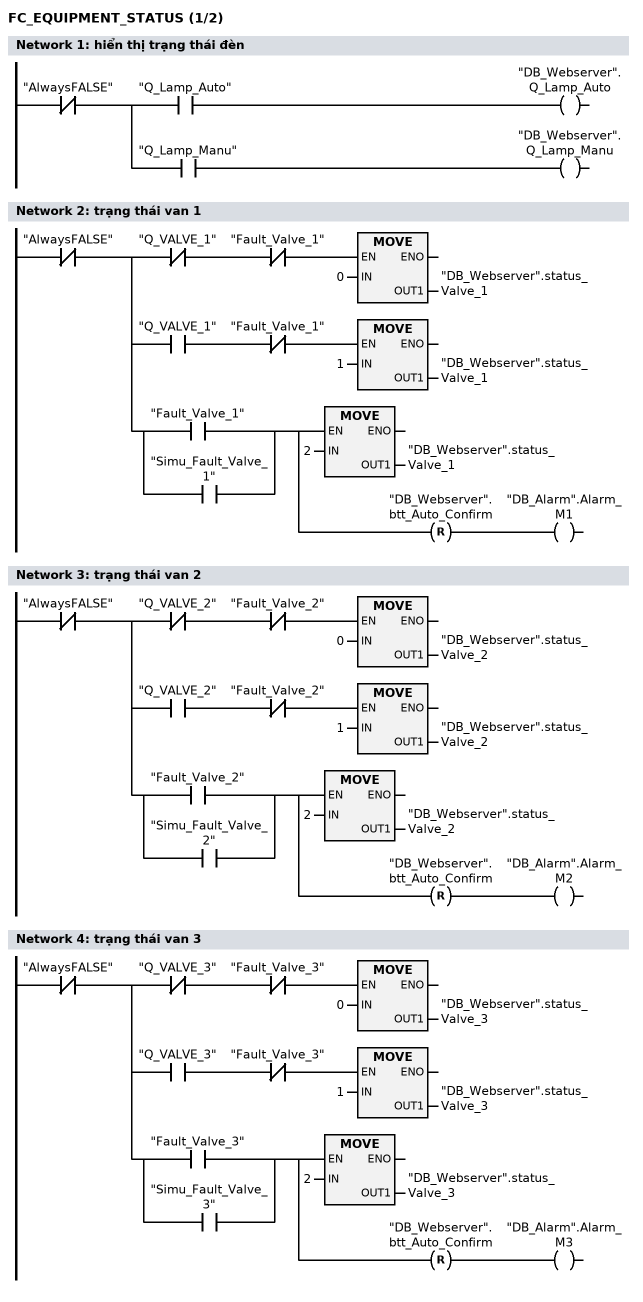
   RUNG wire#powerrail
      I_Contact( "AlwaysFALSE" )
      wire#w1
      Contact( "Q_Lamp_Auto" )
      Coil( "DB_Webserver".Q_Lamp_Auto )
   END_RUNG
   RUNG wire#w1
      Contact( "Q_Lamp_Manu" )
      Coil( "DB_Webserver".Q_Lamp_Manu )
   END_RUNG
   // the same network as SCL:
   "DB_Webserver".Q_Lamp_Auto := NOT "AlwaysFALSE" AND "Q_Lamp_Auto";
   "DB_Webserver".Q_Lamp_Manu := NOT "AlwaysFALSE" AND "Q_Lamp_Manu";
END_REGION

REGION Network 2: trạng thái van 1
   RUNG wire#powerrail
      I_Contact( "AlwaysFALSE" )
      wire#w1
      I_Contact( "Q_VALVE_1" )
      I_Contact( "Fault_Valve_1" )
      Move(in := 0, out1 => "DB_Webserver".status_Valve_1)
   END_RUNG
   RUNG wire#w1
      Contact( "Q_VALVE_1" )
      I_Contact( "Fault_Valve_1" )
      Move(in := 1, out1 => "DB_Webserver".status_Valve_1)
   END_RUNG
   RUNG wire#w1
      Contact( "Fault_Valve_1" )
      wire#w2
      Move(in := 2, out1 => "DB_Webserver".status_Valve_1)
   END_RUNG
   RUNG wire#w1
      Contact( "Simu_Fault_Valve_1" )
   END_RUNG wire#w2
   RUNG wire#w2
      R_Coil( "DB_Webserver".btt_Auto_Confirm )
      Coil( "DB_Alarm".Alarm_M1 )
   END_RUNG
   // the same network as SCL:
   IF NOT "AlwaysFALSE" AND NOT "Q_VALVE_1" AND NOT "Fault_Valve_1" THEN
       "DB_Webserver".status_Valve_1 := 0;
   END_IF;
   IF NOT "AlwaysFALSE" AND "Q_VALVE_1" AND NOT "Fault_Valve_1" THEN
       "DB_Webserver".status_Valve_1 := 1;
   END_IF;
   #_w1 := NOT "AlwaysFALSE" AND ("Fault_Valve_1" OR "Simu_Fault_Valve_1");
   IF #_w1 THEN
       "DB_Webserver".status_Valve_1 := 2;
       "DB_Webserver".btt_Auto_Confirm := FALSE;
   END_IF;
   "DB_Alarm".Alarm_M1 := #_w1;
END_REGION

REGION Network 3: trạng thái van 2
   RUNG wire#powerrail
      I_Contact( "AlwaysFALSE" )
      wire#w1
      I_Contact( "Q_VALVE_2" )
      I_Contact( "Fault_Valve_2" )
      Move(in := 0, out1 => "DB_Webserver".status_Valve_2)
   END_RUNG
   RUNG wire#w1
      Contact( "Q_VALVE_2" )
      I_Contact( "Fault_Valve_2" )
      Move(in := 1, out1 => "DB_Webserver".status_Valve_2)
   END_RUNG
   RUNG wire#w1
      Contact( "Fault_Valve_2" )
      wire#w2
      Move(in := 2, out1 => "DB_Webserver".status_Valve_2)
   END_RUNG
   RUNG wire#w1
      Contact( "Simu_Fault_Valve_2" )
   END_RUNG wire#w2
   RUNG wire#w2
      R_Coil( "DB_Webserver".btt_Auto_Confirm )
      Coil( "DB_Alarm".Alarm_M2 )
   END_RUNG
   // the same network as SCL:
   IF NOT "AlwaysFALSE" AND NOT "Q_VALVE_2" AND NOT "Fault_Valve_2" THEN
       "DB_Webserver".status_Valve_2 := 0;
   END_IF;
   IF NOT "AlwaysFALSE" AND "Q_VALVE_2" AND NOT "Fault_Valve_2" THEN
       "DB_Webserver".status_Valve_2 := 1;
   END_IF;
   #_w1 := NOT "AlwaysFALSE" AND ("Fault_Valve_2" OR "Simu_Fault_Valve_2");
   IF #_w1 THEN
       "DB_Webserver".status_Valve_2 := 2;
       "DB_Webserver".btt_Auto_Confirm := FALSE;
   END_IF;
   "DB_Alarm".Alarm_M2 := #_w1;
END_REGION

REGION Network 4: trạng thái van 3
   RUNG wire#powerrail
      I_Contact( "AlwaysFALSE" )
      wire#w1
      I_Contact( "Q_VALVE_3" )
      I_Contact( "Fault_Valve_3" )
      Move(in := 0, out1 => "DB_Webserver".status_Valve_3)
   END_RUNG
   RUNG wire#w1
      Contact( "Q_VALVE_3" )
      I_Contact( "Fault_Valve_3" )
      Move(in := 1, out1 => "DB_Webserver".status_Valve_3)
   END_RUNG
   RUNG wire#w1
      Contact( "Fault_Valve_3" )
      wire#w2
      Move(in := 2, out1 => "DB_Webserver".status_Valve_3)
   END_RUNG
   RUNG wire#w1
      Contact( "Simu_Fault_Valve_3" )
   END_RUNG wire#w2
   RUNG wire#w2
      R_Coil( "DB_Webserver".btt_Auto_Confirm )
      Coil( "DB_Alarm".Alarm_M3 )
   END_RUNG
   // the same network as SCL:
   IF NOT "AlwaysFALSE" AND NOT "Q_VALVE_3" AND NOT "Fault_Valve_3" THEN
       "DB_Webserver".status_Valve_3 := 0;
   END_IF;
   IF NOT "AlwaysFALSE" AND "Q_VALVE_3" AND NOT "Fault_Valve_3" THEN
       "DB_Webserver".status_Valve_3 := 1;
   END_IF;
   #_w1 := NOT "AlwaysFALSE" AND ("Fault_Valve_3" OR "Simu_Fault_Valve_3");
   IF #_w1 THEN
       "DB_Webserver".status_Valve_3 := 2;
       "DB_Webserver".btt_Auto_Confirm := FALSE;
   END_IF;
   "DB_Alarm".Alarm_M3 := #_w1;
END_REGION

REGION Network 5: trạng thái động cơ
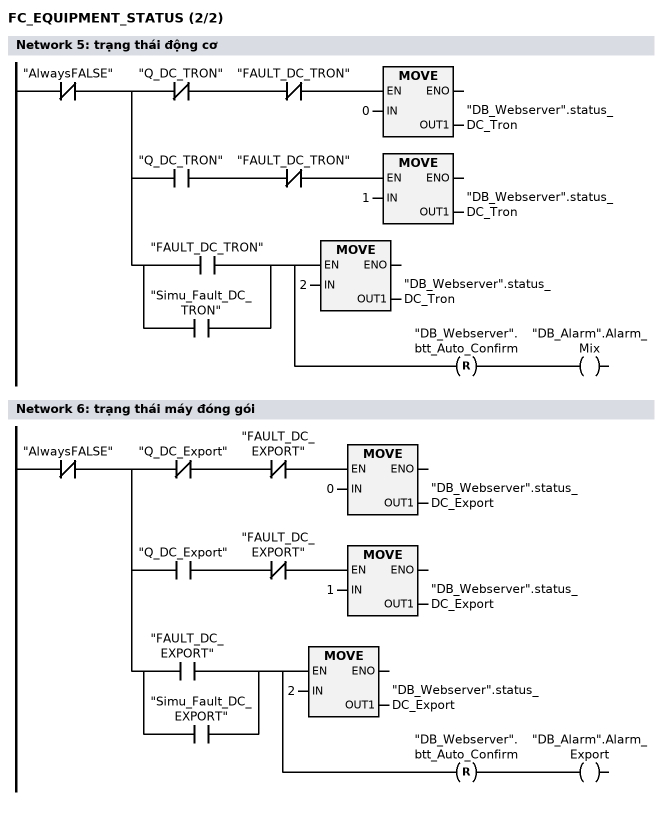
   RUNG wire#powerrail
      I_Contact( "AlwaysFALSE" )
      wire#w1
      I_Contact( "Q_DC_TRON" )
      I_Contact( "FAULT_DC_TRON" )
      Move(in := 0, out1 => "DB_Webserver".status_DC_Tron)
   END_RUNG
   RUNG wire#w1
      Contact( "Q_DC_TRON" )
      I_Contact( "FAULT_DC_TRON" )
      Move(in := 1, out1 => "DB_Webserver".status_DC_Tron)
   END_RUNG
   RUNG wire#w1
      Contact( "FAULT_DC_TRON" )
      wire#w2
      Move(in := 2, out1 => "DB_Webserver".status_DC_Tron)
   END_RUNG
   RUNG wire#w1
      Contact( "Simu_Fault_DC_TRON" )
   END_RUNG wire#w2
   RUNG wire#w2
      R_Coil( "DB_Webserver".btt_Auto_Confirm )
      Coil( "DB_Alarm".Alarm_Mix )
   END_RUNG
   // the same network as SCL:
   IF NOT "AlwaysFALSE" AND NOT "Q_DC_TRON" AND NOT "FAULT_DC_TRON" THEN
       "DB_Webserver".status_DC_Tron := 0;
   END_IF;
   IF NOT "AlwaysFALSE" AND "Q_DC_TRON" AND NOT "FAULT_DC_TRON" THEN
       "DB_Webserver".status_DC_Tron := 1;
   END_IF;
   #_w1 := NOT "AlwaysFALSE" AND ("FAULT_DC_TRON" OR "Simu_Fault_DC_TRON");
   IF #_w1 THEN
       "DB_Webserver".status_DC_Tron := 2;
       "DB_Webserver".btt_Auto_Confirm := FALSE;
   END_IF;
   "DB_Alarm".Alarm_Mix := #_w1;
END_REGION

REGION Network 6: trạng thái máy đóng gói
   RUNG wire#powerrail
      I_Contact( "AlwaysFALSE" )
      wire#w1
      I_Contact( "Q_DC_Export" )
      I_Contact( "FAULT_DC_EXPORT" )
      Move(in := 0, out1 => "DB_Webserver".status_DC_Export)
   END_RUNG
   RUNG wire#w1
      Contact( "Q_DC_Export" )
      I_Contact( "FAULT_DC_EXPORT" )
      Move(in := 1, out1 => "DB_Webserver".status_DC_Export)
   END_RUNG
   RUNG wire#w1
      Contact( "FAULT_DC_EXPORT" )
      wire#w2
      Move(in := 2, out1 => "DB_Webserver".status_DC_Export)
   END_RUNG
   RUNG wire#w1
      Contact( "Simu_Fault_DC_EXPORT" )
   END_RUNG wire#w2
   RUNG wire#w2
      R_Coil( "DB_Webserver".btt_Auto_Confirm )
      Coil( "DB_Alarm".Alarm_Export )
   END_RUNG
   // the same network as SCL:
   IF NOT "AlwaysFALSE" AND NOT "Q_DC_Export" AND NOT "FAULT_DC_EXPORT" THEN
       "DB_Webserver".status_DC_Export := 0;
   END_IF;
   IF NOT "AlwaysFALSE" AND "Q_DC_Export" AND NOT "FAULT_DC_EXPORT" THEN
       "DB_Webserver".status_DC_Export := 1;
   END_IF;
   #_w1 := NOT "AlwaysFALSE" AND ("FAULT_DC_EXPORT" OR "Simu_Fault_DC_EXPORT");
   IF #_w1 THEN
       "DB_Webserver".status_DC_Export := 2;
       "DB_Webserver".btt_Auto_Confirm := FALSE;
   END_IF;
   "DB_Alarm".Alarm_Export := #_w1;
END_REGION
END_FUNCTION

ORGANIZATION_BLOCK "Main"   // OB1, LAD, ProgramCycle
TITLE = "Main Program Sweep (Cycle)"
{ S7_Optimized_Access := 'TRUE' }
VERSION : 0.1
   VAR_INPUT
      Initial_Call : Bool;   // Initial call of this OB
      Remanence : Bool;   // =True, if remanent data are available
   END_VAR
BEGIN

REGION Network 1: chế độ tự động
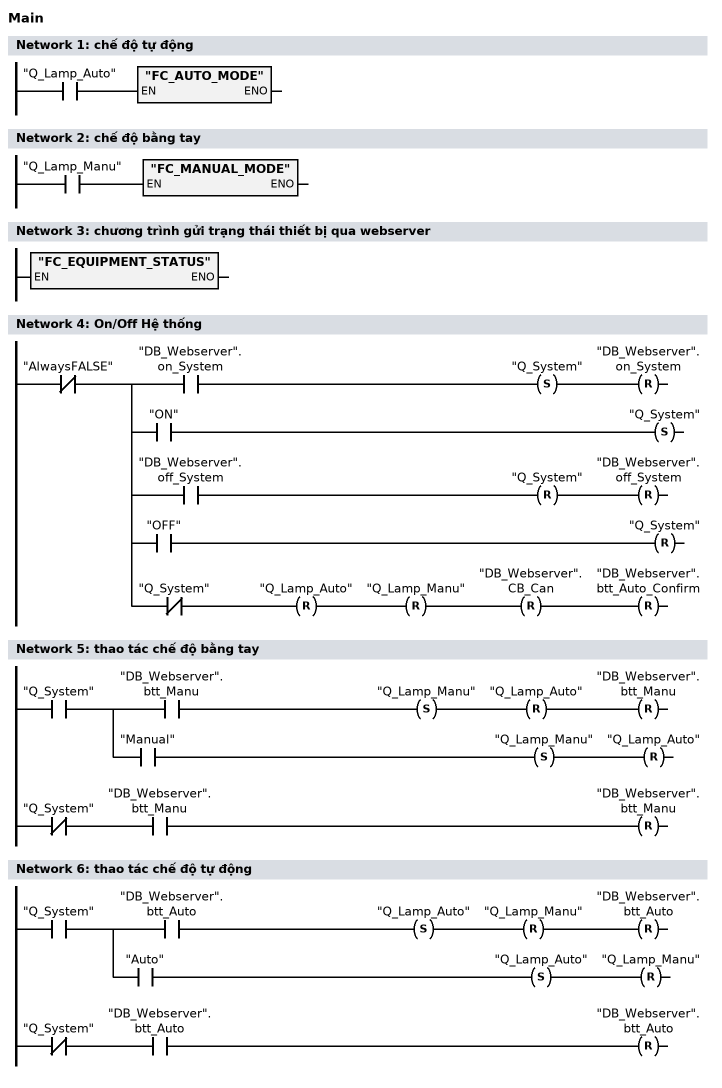
   RUNG wire#powerrail
      Contact( "Q_Lamp_Auto" )
      "FC_AUTO_MODE"()
   END_RUNG
   // the same network as SCL:
   IF "Q_Lamp_Auto" THEN "FC_AUTO_MODE"(); END_IF;
END_REGION

REGION Network 2: chế độ bằng tay
   RUNG wire#powerrail
      Contact( "Q_Lamp_Manu" )
      "FC_MANUAL_MODE"()
   END_RUNG
   // the same network as SCL:
   IF "Q_Lamp_Manu" THEN "FC_MANUAL_MODE"(); END_IF;
END_REGION

REGION Network 3: chương trình gửi trạng thái thiết bị qua webserver
   RUNG wire#powerrail
      "FC_EQUIPMENT_STATUS"()
   END_RUNG
   // the same network as SCL:
   "FC_EQUIPMENT_STATUS"();
END_REGION

REGION Network 4: On/Off Hệ thống
   RUNG wire#powerrail
      I_Contact( "AlwaysFALSE" )
      wire#w1
      Contact( "DB_Webserver".on_System )
      S_Coil( "Q_System" )
      R_Coil( "DB_Webserver".on_System )
   END_RUNG
   RUNG wire#w1
      Contact( "ON" )
      S_Coil( "Q_System" )
   END_RUNG
   RUNG wire#w1
      Contact( "DB_Webserver".off_System )
      R_Coil( "Q_System" )
      R_Coil( "DB_Webserver".off_System )
   END_RUNG
   RUNG wire#w1
      Contact( "OFF" )
      R_Coil( "Q_System" )
   END_RUNG
   RUNG wire#w1
      I_Contact( "Q_System" )
      R_Coil( "Q_Lamp_Auto" )
      R_Coil( "Q_Lamp_Manu" )
      R_Coil( "DB_Webserver".CB_Can )
      R_Coil( "DB_Webserver".btt_Auto_Confirm )
   END_RUNG
   // the same network as SCL:
   IF NOT "AlwaysFALSE" AND "DB_Webserver".on_System THEN
       "Q_System" := TRUE;
       "DB_Webserver".on_System := FALSE;
   END_IF;
   IF NOT "AlwaysFALSE" AND "ON" THEN "Q_System" := TRUE; END_IF;
   IF NOT "AlwaysFALSE" AND "DB_Webserver".off_System THEN
       "Q_System" := FALSE;
       "DB_Webserver".off_System := FALSE;
   END_IF;
   IF NOT "AlwaysFALSE" AND "OFF" THEN "Q_System" := FALSE; END_IF;
   IF NOT "AlwaysFALSE" AND NOT "Q_System" THEN
       "Q_Lamp_Auto" := FALSE;
       "Q_Lamp_Manu" := FALSE;
       "DB_Webserver".CB_Can := FALSE;
       "DB_Webserver".btt_Auto_Confirm := FALSE;
   END_IF;
END_REGION

REGION Network 5: thao tác chế độ bằng tay
   RUNG wire#powerrail
      Contact( "Q_System" )
      wire#w1
      Contact( "DB_Webserver".btt_Manu )
      S_Coil( "Q_Lamp_Manu" )
      R_Coil( "Q_Lamp_Auto" )
      R_Coil( "DB_Webserver".btt_Manu )
   END_RUNG
   RUNG wire#w1
      Contact( "Manual" )
      S_Coil( "Q_Lamp_Manu" )
      R_Coil( "Q_Lamp_Auto" )
   END_RUNG
   RUNG wire#powerrail
      I_Contact( "Q_System" )
      Contact( "DB_Webserver".btt_Manu )
      R_Coil( "DB_Webserver".btt_Manu )
   END_RUNG
   // the same network as SCL:
   IF "Q_System" AND "DB_Webserver".btt_Manu THEN
       "Q_Lamp_Manu" := TRUE;
       "Q_Lamp_Auto" := FALSE;
       "DB_Webserver".btt_Manu := FALSE;
   END_IF;
   IF "Q_System" AND "Manual" THEN
       "Q_Lamp_Manu" := TRUE;
       "Q_Lamp_Auto" := FALSE;
   END_IF;
   IF NOT "Q_System" AND "DB_Webserver".btt_Manu THEN "DB_Webserver".btt_Manu := FALSE; END_IF;
END_REGION

REGION Network 6: thao tác chế độ tự động
   RUNG wire#powerrail
      Contact( "Q_System" )
      wire#w1
      Contact( "DB_Webserver".btt_Auto )
      S_Coil( "Q_Lamp_Auto" )
      R_Coil( "Q_Lamp_Manu" )
      R_Coil( "DB_Webserver".btt_Auto )
   END_RUNG
   RUNG wire#w1
      Contact( "Auto" )
      S_Coil( "Q_Lamp_Auto" )
      R_Coil( "Q_Lamp_Manu" )
   END_RUNG
   RUNG wire#powerrail
      I_Contact( "Q_System" )
      Contact( "DB_Webserver".btt_Auto )
      R_Coil( "DB_Webserver".btt_Auto )
   END_RUNG
   // the same network as SCL:
   IF "Q_System" AND "DB_Webserver".btt_Auto THEN
       "Q_Lamp_Auto" := TRUE;
       "Q_Lamp_Manu" := FALSE;
       "DB_Webserver".btt_Auto := FALSE;
   END_IF;
   IF "Q_System" AND "Auto" THEN
       "Q_Lamp_Auto" := TRUE;
       "Q_Lamp_Manu" := FALSE;
   END_IF;
   IF NOT "Q_System" AND "DB_Webserver".btt_Auto THEN "DB_Webserver".btt_Auto := FALSE; END_IF;
END_REGION
END_ORGANIZATION_BLOCK

// ===== PLC "STATION_2"  CPU 1215C DC/DC/DC =====

VAR_GLOBAL   // PLC tag table "Default tag table"
   "Clock_Byte" AT %MB0 : Byte;
   "Clock_10Hz" AT %M0.0 : Bool;
   "Clock_5Hz" AT %M0.1 : Bool;
   "Clock_2.5Hz" AT %M0.2 : Bool;
   "Clock_2Hz" AT %M0.3 : Bool;
   "Clock_1.25Hz" AT %M0.4 : Bool;
   "Clock_1Hz" AT %M0.5 : Bool;
   "Clock_0.625Hz" AT %M0.6 : Bool;
   "Clock_0.5Hz" AT %M0.7 : Bool;
   "System_Byte" AT %MB1 : Byte;
   "FirstScan" AT %M1.0 : Bool;
   "DiagStatusUpdate" AT %M1.1 : Bool;
   "AlwaysTRUE" AT %M1.2 : Bool;
   "AlwaysFALSE" AT %M1.3 : Bool;
   "XUNG_PTRIG_1" AT %M10.0 : Bool;
   "XUNG_PTRIG_2" AT %M10.1 : Bool;
   "XUNG_PTRIG_3" AT %M10.2 : Bool;
   "XUNG_PTRIG_4" AT %M10.3 : Bool;
   "XUNG_PTRIG_5" AT %M10.4 : Bool;
   "XUNG_PTRIG_6" AT %M10.5 : Bool;
   "XUNG_PTRIG_7" AT %M10.6 : Bool;
   "XUNG_PTRIG_8" AT %M10.7 : Bool;
END_VAR

VAR_GLOBAL   // PLC tag table "Input"
   "Fault_Valve_1" AT %I0.0 : Bool;   // Bit báo lỗi van 1
   "Fault_Valve_2" AT %I0.1 : Bool;   // Bit báo lỗi van 2
   "Fault_Valve_3" AT %I0.2 : Bool;   // Bit báo lỗi van 3
   "FAULT_DC_TRON" AT %I0.3 : Bool;   // Bit báo lỗi động cơ trộn
   "Auto" AT %I0.5 : Bool;   // Chế độ Auto
   "Manual" AT %I0.6 : Bool;   // Chế độ Manual
   "FAULT_DC_EXPORT" AT %I0.4 : Bool;   // Bit baso lỗi máy đóng gói
   "ON" AT %I0.7 : Bool;   // Bật Hệ thống
   "OFF" AT %I1.0 : Bool;   // Tắt hệ thống
END_VAR

VAR_GLOBAL   // PLC tag table "Output"
   "Q_VALVE_1" AT %Q0.0 : Bool;   // Đầu ra van 1
   "Q_VALVE_2" AT %Q0.1 : Bool;   // Đầu ra van 2
   "Q_VALVE_3" AT %Q0.2 : Bool;   // Đầu ra van 3
   "Q_DC_TRON" AT %Q0.3 : Bool;   // Đầu ra động cơ trộn
   "Q_Lamp_Auto" AT %Q0.5 : Bool;
   "Q_Lamp_Manu" AT %Q0.6 : Bool;
   "Q_DC_Export" AT %Q0.4 : Bool;   // Đầu ra máy đóng gói
   "Q_System" AT %Q0.7 : Bool;
END_VAR

VAR_GLOBAL   // PLC tag table "simulation"
   "Simu_Fault_Valve_1" AT %M20.0 : Bool;
   "Simu_Fault_Valve_2" AT %M20.1 : Bool;
   "Simu_Fault_Valve_3" AT %M20.2 : Bool;
   "Simu_Fault_DC_TRON" AT %M20.3 : Bool;
   "Simu_Fault_DC_EXPORT" AT %M20.4 : Bool;
END_VAR

DATA_BLOCK "DB_Webserver"   // DB1
{ S7_Optimized_Access := 'FALSE' }
VERSION : 0.1
   VAR
      btt_Auto : Bool;   // Nút nhấn chế độ tự động
      btt_Manu : Bool;   // Nút nhấn chế độ bằng tay
      btt_Auto_Confirm : Bool;   // Nút nhấn xác nhận
      btt_V1_Open : Bool;   // Nút nhấn chế độ bằng tay mở van 1
      btt_V1_Close : Bool;   // Nút nhấn chế độ bằng tay đóng van 1
      btt_V2_Open : Bool;   // Nút nhấn chế độ bằng tay mở van 2
      btt_V2_Close : Bool;   // Nút nhấn chế độ bằng tay đóng van 2
      btt_V3_Open : Bool;   // Nút nhấn chế độ bằng tay mở van 3
      btt_V3_Close : Bool;   // Nút nhấn chế độ bằng tay đóng van 3
      btt_DC_Tron_Run : Bool;   // Nút nhấn chế độ bằng tay chạy ĐC trộn
      btt_DC_Tron_Stop : Bool;   // Nút nhấn chế độ bằng tay dừng ĐC trộn
      btt_DC_Export_Run : Bool;   // Nút nhấn chế độ bằng tay chạy máy đóng gói
      btt_DC_Export_Stop : Bool;   // Nút nhấn chế độ bằng tay đóng máy đóng gói
      CB_Can : Bool;   // Cảm biến cạn bồn trộn
      Q_Lamp_Auto : Bool;   // Đèn chế độ tự động
      Q_Lamp_Manu : Bool;   // Đèn chế độ bằng tay
      status_Valve_1 : Byte;   // Trạng thái van 1 (0 = Đang đóng, 1 = Đang mở, 2 = Đang lỗi)
      status_Valve_2 : Byte;   // Trạng thái van 2 (0 = Đang đóng, 1 = Đang mở, 2 = Đang lỗi)
      status_Valve_3 : Byte;   // Trạng thái van 3 (0 = Đang đóng, 1 = Đang mở, 2 = Đang lỗi)
      status_DC_Tron : Byte;   // Trạng thái ĐC trộn (0 = Đang đóng, 1 = Đang mở, 2 = Đang lỗi)
      status_DC_Export : Byte;   // Trạng thái Máy đóng gói (0 = Đang đóng, 1 = Đang mở, 2 = Đang lỗi)
      Setting_Time_Tron : Int := 10;   // Cài đặt thời gian trộn
      Act_Time_Tron : Int;   // Giá trị thực tế thời gian trộn
      Setting_Weight_1 : Real := 12.25;   // Cài đặt trọng lượng liệu 1
      Setting_Weight_2 : Real := 20.45;   // Cài đặt trọng lượng liệu 2
      Setting_Weight_3 : Real := 10.12;   // Cài đặt trọng lượng liệu 3
      Act_Weight_1 : Real;   // Giá trị thực tế trọng lượng liệu 1
      Act_Weight_2 : Real;   // Giá trị thực tế trọng lượng liệu 2
      Act_Weight_3 : Real;   // Giá trị thực tế trọng lượng liệu 3
      sql_insert_Trigger : Bool;   // Bit lưu giá trị lên SQL
      sql_insert_On : Bool;
      sql_insert_Off : Bool;
      sql_insert_Temp : Bool;
      sql_delete_Trigger : Bool;   // Bit xóa dữ liệu SQL
      sql_OrderID : String := 'Product 0';   // ID đơn hàng cần trộn
      sql_Weight1_Setting : Real;
      sql_Weight2_Setting : Real;
      sql_Weight3_Setting : Real;
      sql_Weight1_Actual : Real;
      sql_Weight2_Actual : Real;
      sql_Weight3_Actual : Real;
      sql_Time_Tron_Setting : Int;
      sql_Time_Tron_Actual : Int;
      on_System : Bool;
      off_System : Bool;
   END_VAR
BEGIN
END_DATA_BLOCK

DATA_BLOCK "Data"   // DB2
{ S7_Optimized_Access := 'TRUE' }
VERSION : 0.1
   VAR
      act_Step_1 : Bool;   // Giá trị thực tế bước 1
      act_Step_2 : Bool;   // Giá trị thực tế bước 2
      act_Step_3 : Bool;   // Giá trị thực tế bước 3
      act_done_valve_1 : Bool;   // Bit báo đã xả xong nguyên liệu 1
      act_done_valve_2 : Bool;   // Bit báo đã xả xong nguyên liệu 2
      act_done_valve_3 : Bool;   // Bit báo đã xả xong nguyên liệu 3
   END_VAR
BEGIN
END_DATA_BLOCK

DATA_BLOCK "DB_Alarm"   // DB4
{ S7_Optimized_Access := 'FALSE' }
VERSION : 0.1
   VAR
      Alarm_M1 : Bool;
      Alarm_M2 : Bool;
      Alarm_M3 : Bool;
      Alarm_Mix : Bool;
      Alarm_Export : Bool;
   END_VAR
BEGIN
END_DATA_BLOCK

// folder: System blocks/Program resources

DATA_BLOCK "TIMER_SIMU"   // DB3
{ S7_Optimized_Access := 'TRUE' }
AUTHOR : Simatic
FAMILY : IEC
NAME : IEC_TMR
VERSION : 1.0
// stored: InstanceOfName IEC_TIMER
"IEC_TIMER"
BEGIN
END_DATA_BLOCK

DATA_BLOCK "TImer_SQL_Delete"   // DB5
{ S7_Optimized_Access := 'TRUE' }
AUTHOR : Simatic
FAMILY : IEC
NAME : IEC_TMR
VERSION : 1.0
// stored: InstanceOfName IEC_TIMER
"IEC_TIMER"
BEGIN
END_DATA_BLOCK

DATA_BLOCK "sql_insert_on"   // DB6
{ S7_Optimized_Access := 'TRUE' }
AUTHOR : Simatic
FAMILY : IEC
NAME : IEC_TMR
VERSION : 1.0
// stored: InstanceOfName IEC_TIMER
"IEC_TIMER"
BEGIN
END_DATA_BLOCK

// folder: (top level)

FUNCTION "FC_MANUAL_MODE" : Void   // FC1, LAD
{ S7_Optimized_Access := 'TRUE' }
VERSION : 0.1
   VAR_TEMP   // added for the SCL form of the ladder/FBD networks
      _w1 : Bool;
      _w2 : Bool;
      _w3 : Bool;
      _w4 : Bool;
      _w5 : Bool;
      _w6 : Bool;
   END_VAR
BEGIN

REGION Network 1: Đầu ra động cơ trộn
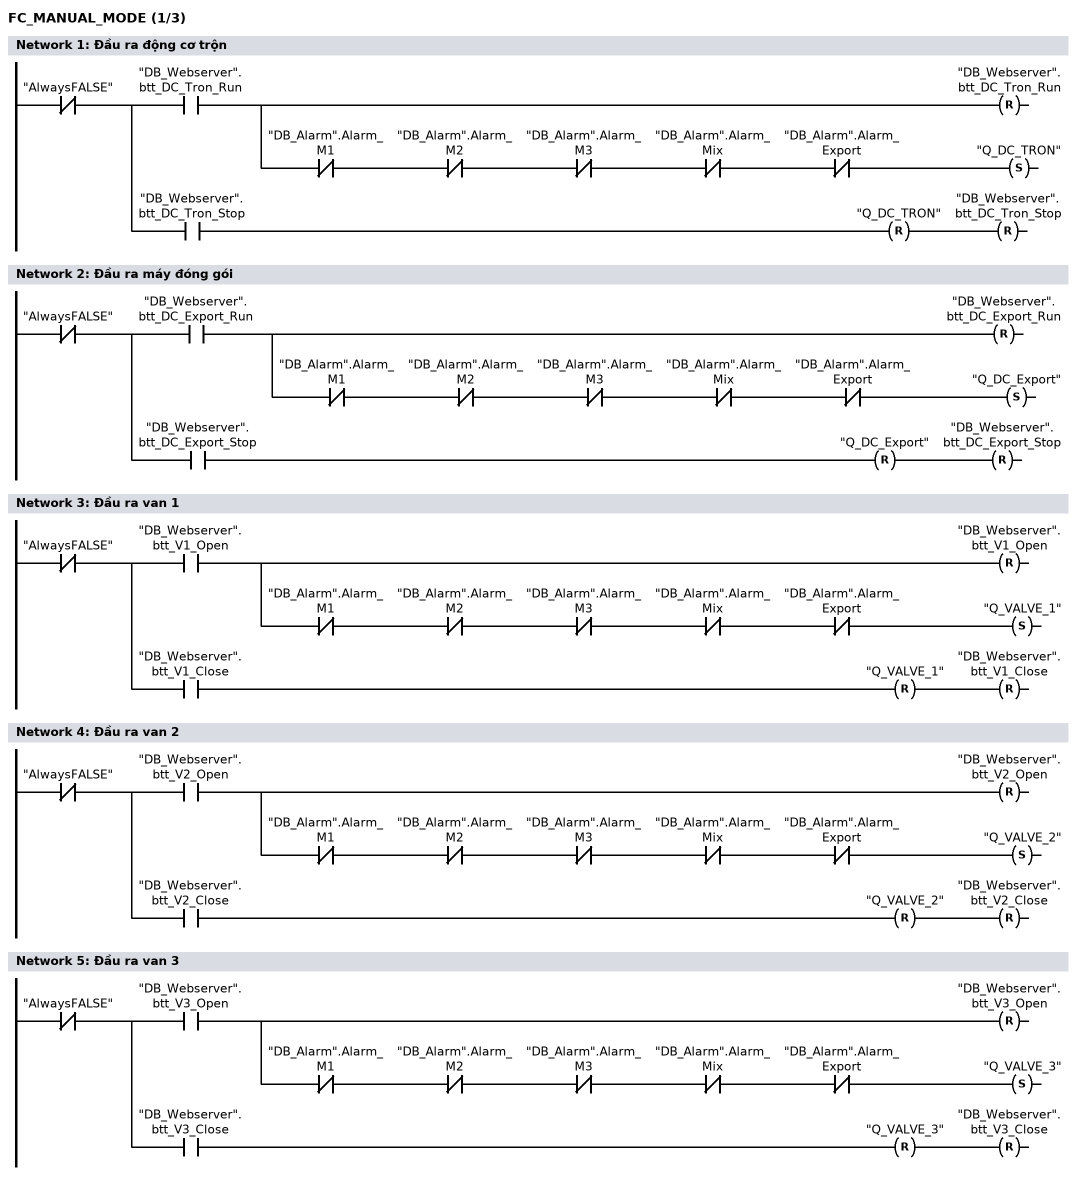
   RUNG wire#powerrail
      I_Contact( "AlwaysFALSE" )
      wire#w1
      Contact( "DB_Webserver".btt_DC_Tron_Run )
      wire#w2
      R_Coil( "DB_Webserver".btt_DC_Tron_Run )
   END_RUNG
   RUNG wire#w2
      I_Contact( "DB_Alarm".Alarm_M1 )
      I_Contact( "DB_Alarm".Alarm_M2 )
      I_Contact( "DB_Alarm".Alarm_M3 )
      I_Contact( "DB_Alarm".Alarm_Mix )
      I_Contact( "DB_Alarm".Alarm_Export )
      S_Coil( "Q_DC_TRON" )
   END_RUNG
   RUNG wire#w1
      Contact( "DB_Webserver".btt_DC_Tron_Stop )
      R_Coil( "Q_DC_TRON" )
      R_Coil( "DB_Webserver".btt_DC_Tron_Stop )
   END_RUNG
   // the same network as SCL:
   #_w1 := NOT "AlwaysFALSE" AND "DB_Webserver".btt_DC_Tron_Run;
   IF #_w1 THEN "DB_Webserver".btt_DC_Tron_Run := FALSE; END_IF;
   IF #_w1 AND NOT "DB_Alarm".Alarm_M1 AND NOT "DB_Alarm".Alarm_M2 AND NOT "DB_Alarm".Alarm_M3 AND NOT "DB_Alarm".Alarm_Mix AND NOT "DB_Alarm".Alarm_Export THEN
       "Q_DC_TRON" := TRUE;
   END_IF;
   IF NOT "AlwaysFALSE" AND "DB_Webserver".btt_DC_Tron_Stop THEN
       "Q_DC_TRON" := FALSE;
       "DB_Webserver".btt_DC_Tron_Stop := FALSE;
   END_IF;
END_REGION

REGION Network 2: Đầu ra máy đóng gói
   RUNG wire#powerrail
      I_Contact( "AlwaysFALSE" )
      wire#w1
      Contact( "DB_Webserver".btt_DC_Export_Run )
      wire#w2
      R_Coil( "DB_Webserver".btt_DC_Export_Run )
   END_RUNG
   RUNG wire#w2
      I_Contact( "DB_Alarm".Alarm_M1 )
      I_Contact( "DB_Alarm".Alarm_M2 )
      I_Contact( "DB_Alarm".Alarm_M3 )
      I_Contact( "DB_Alarm".Alarm_Mix )
      I_Contact( "DB_Alarm".Alarm_Export )
      S_Coil( "Q_DC_Export" )
   END_RUNG
   RUNG wire#w1
      Contact( "DB_Webserver".btt_DC_Export_Stop )
      R_Coil( "Q_DC_Export" )
      R_Coil( "DB_Webserver".btt_DC_Export_Stop )
   END_RUNG
   // the same network as SCL:
   #_w1 := NOT "AlwaysFALSE" AND "DB_Webserver".btt_DC_Export_Run;
   IF #_w1 THEN "DB_Webserver".btt_DC_Export_Run := FALSE; END_IF;
   IF #_w1 AND NOT "DB_Alarm".Alarm_M1 AND NOT "DB_Alarm".Alarm_M2 AND NOT "DB_Alarm".Alarm_M3 AND NOT "DB_Alarm".Alarm_Mix AND NOT "DB_Alarm".Alarm_Export THEN
       "Q_DC_Export" := TRUE;
   END_IF;
   IF NOT "AlwaysFALSE" AND "DB_Webserver".btt_DC_Export_Stop THEN
       "Q_DC_Export" := FALSE;
       "DB_Webserver".btt_DC_Export_Stop := FALSE;
   END_IF;
END_REGION

REGION Network 3: Đầu ra van 1
   RUNG wire#powerrail
      I_Contact( "AlwaysFALSE" )
      wire#w1
      Contact( "DB_Webserver".btt_V1_Open )
      wire#w2
      R_Coil( "DB_Webserver".btt_V1_Open )
   END_RUNG
   RUNG wire#w2
      I_Contact( "DB_Alarm".Alarm_M1 )
      I_Contact( "DB_Alarm".Alarm_M2 )
      I_Contact( "DB_Alarm".Alarm_M3 )
      I_Contact( "DB_Alarm".Alarm_Mix )
      I_Contact( "DB_Alarm".Alarm_Export )
      S_Coil( "Q_VALVE_1" )
   END_RUNG
   RUNG wire#w1
      Contact( "DB_Webserver".btt_V1_Close )
      R_Coil( "Q_VALVE_1" )
      R_Coil( "DB_Webserver".btt_V1_Close )
   END_RUNG
   // the same network as SCL:
   #_w1 := NOT "AlwaysFALSE" AND "DB_Webserver".btt_V1_Open;
   IF #_w1 THEN "DB_Webserver".btt_V1_Open := FALSE; END_IF;
   IF #_w1 AND NOT "DB_Alarm".Alarm_M1 AND NOT "DB_Alarm".Alarm_M2 AND NOT "DB_Alarm".Alarm_M3 AND NOT "DB_Alarm".Alarm_Mix AND NOT "DB_Alarm".Alarm_Export THEN
       "Q_VALVE_1" := TRUE;
   END_IF;
   IF NOT "AlwaysFALSE" AND "DB_Webserver".btt_V1_Close THEN
       "Q_VALVE_1" := FALSE;
       "DB_Webserver".btt_V1_Close := FALSE;
   END_IF;
END_REGION

REGION Network 4: Đầu ra van 2
   RUNG wire#powerrail
      I_Contact( "AlwaysFALSE" )
      wire#w1
      Contact( "DB_Webserver".btt_V2_Open )
      wire#w2
      R_Coil( "DB_Webserver".btt_V2_Open )
   END_RUNG
   RUNG wire#w2
      I_Contact( "DB_Alarm".Alarm_M1 )
      I_Contact( "DB_Alarm".Alarm_M2 )
      I_Contact( "DB_Alarm".Alarm_M3 )
      I_Contact( "DB_Alarm".Alarm_Mix )
      I_Contact( "DB_Alarm".Alarm_Export )
      S_Coil( "Q_VALVE_2" )
   END_RUNG
   RUNG wire#w1
      Contact( "DB_Webserver".btt_V2_Close )
      R_Coil( "Q_VALVE_2" )
      R_Coil( "DB_Webserver".btt_V2_Close )
   END_RUNG
   // the same network as SCL:
   #_w1 := NOT "AlwaysFALSE" AND "DB_Webserver".btt_V2_Open;
   IF #_w1 THEN "DB_Webserver".btt_V2_Open := FALSE; END_IF;
   IF #_w1 AND NOT "DB_Alarm".Alarm_M1 AND NOT "DB_Alarm".Alarm_M2 AND NOT "DB_Alarm".Alarm_M3 AND NOT "DB_Alarm".Alarm_Mix AND NOT "DB_Alarm".Alarm_Export THEN
       "Q_VALVE_2" := TRUE;
   END_IF;
   IF NOT "AlwaysFALSE" AND "DB_Webserver".btt_V2_Close THEN
       "Q_VALVE_2" := FALSE;
       "DB_Webserver".btt_V2_Close := FALSE;
   END_IF;
END_REGION

REGION Network 5: Đầu ra van 3
   RUNG wire#powerrail
      I_Contact( "AlwaysFALSE" )
      wire#w1
      Contact( "DB_Webserver".btt_V3_Open )
      wire#w2
      R_Coil( "DB_Webserver".btt_V3_Open )
   END_RUNG
   RUNG wire#w2
      I_Contact( "DB_Alarm".Alarm_M1 )
      I_Contact( "DB_Alarm".Alarm_M2 )
      I_Contact( "DB_Alarm".Alarm_M3 )
      I_Contact( "DB_Alarm".Alarm_Mix )
      I_Contact( "DB_Alarm".Alarm_Export )
      S_Coil( "Q_VALVE_3" )
   END_RUNG
   RUNG wire#w1
      Contact( "DB_Webserver".btt_V3_Close )
      R_Coil( "Q_VALVE_3" )
      R_Coil( "DB_Webserver".btt_V3_Close )
   END_RUNG
   // the same network as SCL:
   #_w1 := NOT "AlwaysFALSE" AND "DB_Webserver".btt_V3_Open;
   IF #_w1 THEN "DB_Webserver".btt_V3_Open := FALSE; END_IF;
   IF #_w1 AND NOT "DB_Alarm".Alarm_M1 AND NOT "DB_Alarm".Alarm_M2 AND NOT "DB_Alarm".Alarm_M3 AND NOT "DB_Alarm".Alarm_Mix AND NOT "DB_Alarm".Alarm_Export THEN
       "Q_VALVE_3" := TRUE;
   END_IF;
   IF NOT "AlwaysFALSE" AND "DB_Webserver".btt_V3_Close THEN
       "Q_VALVE_3" := FALSE;
       "DB_Webserver".btt_V3_Close := FALSE;
   END_IF;
END_REGION

REGION Network 6: mô phỏng tăng trọng lượng
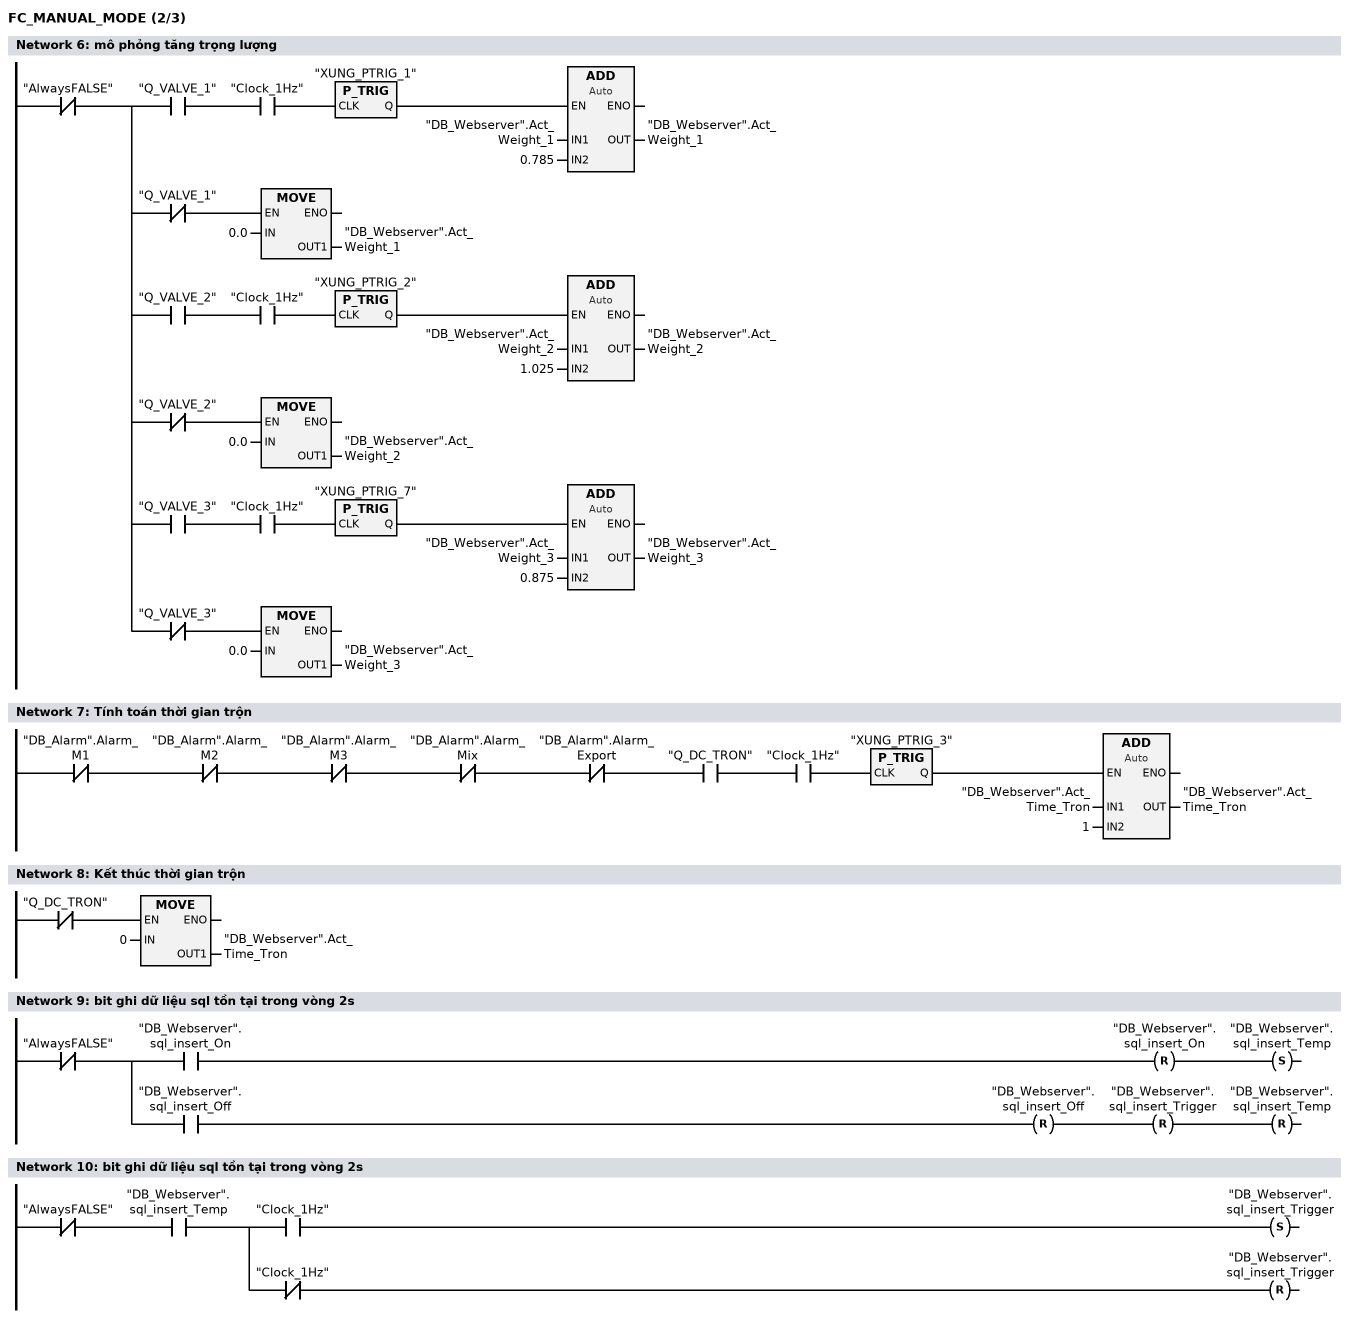
   RUNG wire#powerrail
      I_Contact( "AlwaysFALSE" )
      wire#w1
      Contact( "Q_VALVE_1" )
      Contact( "Clock_1Hz" )
      P_Trig( "XUNG_PTRIG_1" )
      Add(in1 := "DB_Webserver".Act_Weight_1, in2 := 0.785, out => "DB_Webserver".Act_Weight_1)
   END_RUNG
   RUNG wire#w1
      I_Contact( "Q_VALVE_1" )
      Move(in := 0.0, out1 => "DB_Webserver".Act_Weight_1)
   END_RUNG
   RUNG wire#w1
      Contact( "Q_VALVE_2" )
      Contact( "Clock_1Hz" )
      P_Trig( "XUNG_PTRIG_2" )
      Add(in1 := "DB_Webserver".Act_Weight_2, in2 := 1.025, out => "DB_Webserver".Act_Weight_2)
   END_RUNG
   RUNG wire#w1
      I_Contact( "Q_VALVE_2" )
      Move(in := 0.0, out1 => "DB_Webserver".Act_Weight_2)
   END_RUNG
   RUNG wire#w1
      Contact( "Q_VALVE_3" )
      Contact( "Clock_1Hz" )
      P_Trig( "XUNG_PTRIG_7" )
      Add(in1 := "DB_Webserver".Act_Weight_3, in2 := 0.875, out => "DB_Webserver".Act_Weight_3)
   END_RUNG
   RUNG wire#w1
      I_Contact( "Q_VALVE_3" )
      Move(in := 0.0, out1 => "DB_Webserver".Act_Weight_3)
   END_RUNG
   // the same network as SCL:
   #_w1 := NOT "AlwaysFALSE" AND "Q_VALVE_1" AND "Clock_1Hz";
   #_w2 := #_w1 AND NOT "XUNG_PTRIG_1";   // rising edge
   "XUNG_PTRIG_1" := #_w1;
   IF #_w2 THEN "DB_Webserver".Act_Weight_1 := "DB_Webserver".Act_Weight_1 + 0.785; END_IF;
   IF NOT "AlwaysFALSE" AND NOT "Q_VALVE_1" THEN "DB_Webserver".Act_Weight_1 := 0.0; END_IF;
   #_w3 := NOT "AlwaysFALSE" AND "Q_VALVE_2" AND "Clock_1Hz";
   #_w4 := #_w3 AND NOT "XUNG_PTRIG_2";   // rising edge
   "XUNG_PTRIG_2" := #_w3;
   IF #_w4 THEN "DB_Webserver".Act_Weight_2 := "DB_Webserver".Act_Weight_2 + 1.025; END_IF;
   IF NOT "AlwaysFALSE" AND NOT "Q_VALVE_2" THEN "DB_Webserver".Act_Weight_2 := 0.0; END_IF;
   #_w5 := NOT "AlwaysFALSE" AND "Q_VALVE_3" AND "Clock_1Hz";
   #_w6 := #_w5 AND NOT "XUNG_PTRIG_7";   // rising edge
   "XUNG_PTRIG_7" := #_w5;
   IF #_w6 THEN "DB_Webserver".Act_Weight_3 := "DB_Webserver".Act_Weight_3 + 0.875; END_IF;
   IF NOT "AlwaysFALSE" AND NOT "Q_VALVE_3" THEN "DB_Webserver".Act_Weight_3 := 0.0; END_IF;
END_REGION

REGION Network 7: Tính toán thời gian trộn
   RUNG wire#powerrail
      I_Contact( "DB_Alarm".Alarm_M1 )
      I_Contact( "DB_Alarm".Alarm_M2 )
      I_Contact( "DB_Alarm".Alarm_M3 )
      I_Contact( "DB_Alarm".Alarm_Mix )
      I_Contact( "DB_Alarm".Alarm_Export )
      Contact( "Q_DC_TRON" )
      Contact( "Clock_1Hz" )
      P_Trig( "XUNG_PTRIG_3" )
      Add(in1 := "DB_Webserver".Act_Time_Tron, in2 := 1, out => "DB_Webserver".Act_Time_Tron)
   END_RUNG
   // the same network as SCL:
   #_w1 := NOT "DB_Alarm".Alarm_M1 AND NOT "DB_Alarm".Alarm_M2 AND NOT "DB_Alarm".Alarm_M3 AND NOT "DB_Alarm".Alarm_Mix AND NOT "DB_Alarm".Alarm_Export AND "Q_DC_TRON" AND "Clock_1Hz";
   #_w2 := #_w1 AND NOT "XUNG_PTRIG_3";   // rising edge
   "XUNG_PTRIG_3" := #_w1;
   IF #_w2 THEN "DB_Webserver".Act_Time_Tron := "DB_Webserver".Act_Time_Tron + 1; END_IF;
END_REGION

REGION Network 8: Kết thúc thời gian trộn
   RUNG wire#powerrail
      I_Contact( "Q_DC_TRON" )
      Move(in := 0, out1 => "DB_Webserver".Act_Time_Tron)
   END_RUNG
   // the same network as SCL:
   IF NOT "Q_DC_TRON" THEN "DB_Webserver".Act_Time_Tron := 0; END_IF;
END_REGION

REGION Network 9: bit ghi dữ liệu sql tồn tại trong vòng 2s
   RUNG wire#powerrail
      I_Contact( "AlwaysFALSE" )
      wire#w1
      Contact( "DB_Webserver".sql_insert_On )
      R_Coil( "DB_Webserver".sql_insert_On )
      S_Coil( "DB_Webserver".sql_insert_Temp )
   END_RUNG
   RUNG wire#w1
      Contact( "DB_Webserver".sql_insert_Off )
      R_Coil( "DB_Webserver".sql_insert_Off )
      R_Coil( "DB_Webserver".sql_insert_Trigger )
      R_Coil( "DB_Webserver".sql_insert_Temp )
   END_RUNG
   // the same network as SCL:
   #_w1 := NOT "AlwaysFALSE" AND "DB_Webserver".sql_insert_On;
   IF #_w1 THEN
       "DB_Webserver".sql_insert_On := FALSE;
       "DB_Webserver".sql_insert_Temp := TRUE;
   END_IF;
   #_w2 := NOT "AlwaysFALSE" AND "DB_Webserver".sql_insert_Off;
   IF #_w2 THEN
       "DB_Webserver".sql_insert_Off := FALSE;
       "DB_Webserver".sql_insert_Trigger := FALSE;
       "DB_Webserver".sql_insert_Temp := FALSE;
   END_IF;
END_REGION

REGION Network 10: bit ghi dữ liệu sql tồn tại trong vòng 2s
   RUNG wire#powerrail
      I_Contact( "AlwaysFALSE" )
      Contact( "DB_Webserver".sql_insert_Temp )
      wire#w1
      Contact( "Clock_1Hz" )
      S_Coil( "DB_Webserver".sql_insert_Trigger )
   END_RUNG
   RUNG wire#w1
      I_Contact( "Clock_1Hz" )
      R_Coil( "DB_Webserver".sql_insert_Trigger )
   END_RUNG
   // the same network as SCL:
   #_w1 := NOT "AlwaysFALSE" AND "DB_Webserver".sql_insert_Temp;
   IF #_w1 AND "Clock_1Hz" THEN "DB_Webserver".sql_insert_Trigger := TRUE; END_IF;
   IF #_w1 AND NOT "Clock_1Hz" THEN "DB_Webserver".sql_insert_Trigger := FALSE; END_IF;
END_REGION

REGION Network 11: bit ghi dữ liệu sql tồn tại trong vòng 2s
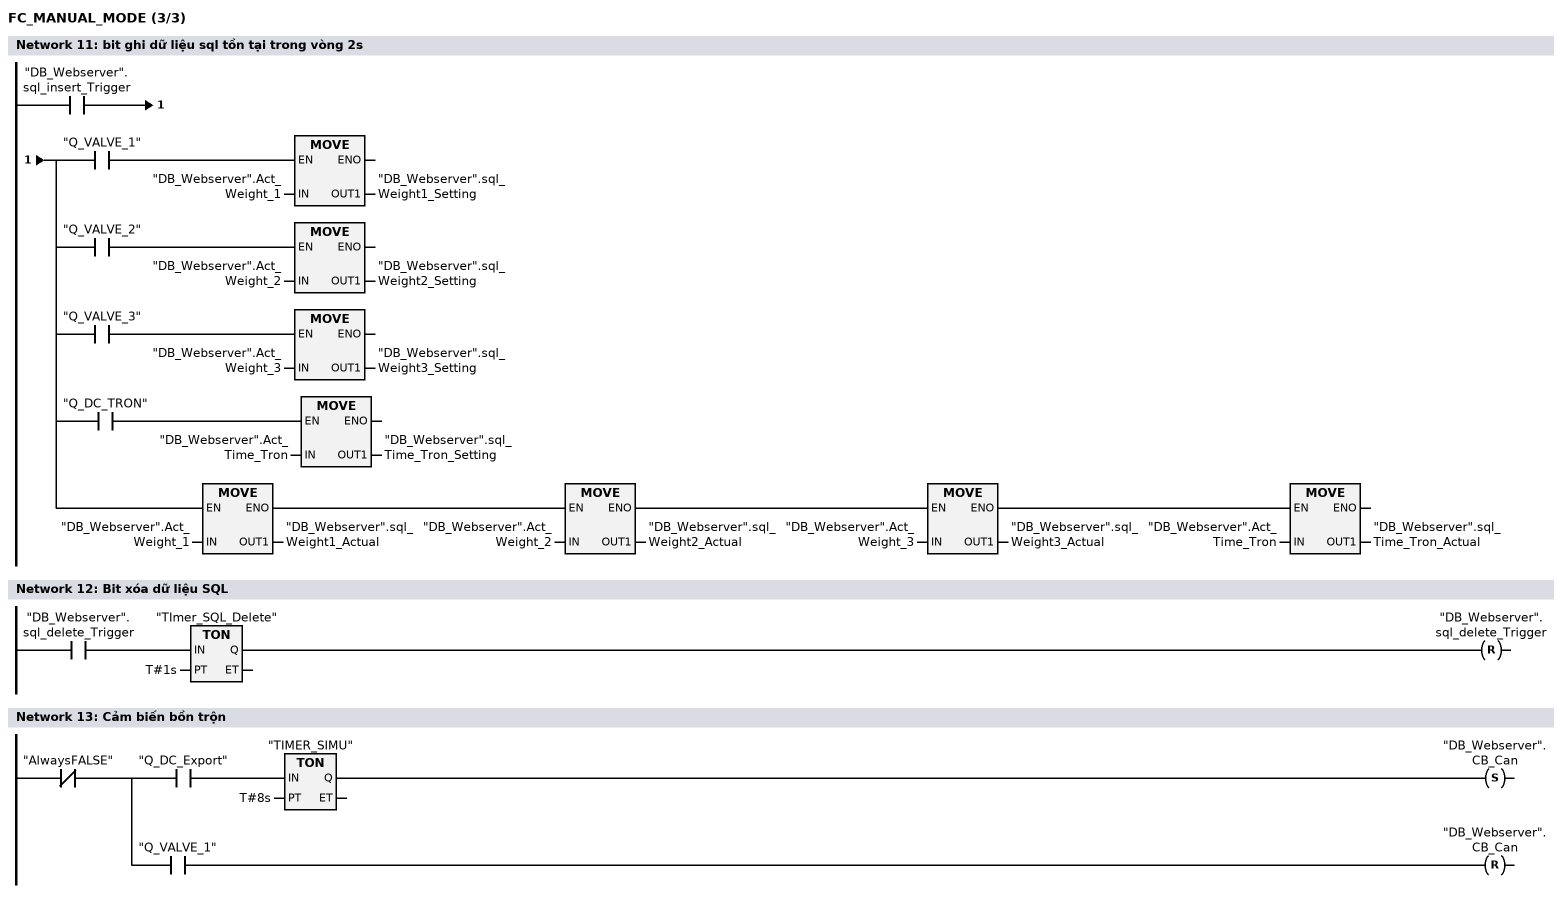
   RUNG wire#powerrail
      Contact( "DB_Webserver".sql_insert_Trigger )
      wire#w1
      Contact( "Q_VALVE_1" )
      Move(in := "DB_Webserver".Act_Weight_1, out1 => "DB_Webserver".sql_Weight1_Setting)
   END_RUNG
   RUNG wire#w1
      Contact( "Q_VALVE_2" )
      Move(in := "DB_Webserver".Act_Weight_2, out1 => "DB_Webserver".sql_Weight2_Setting)
   END_RUNG
   RUNG wire#w1
      Contact( "Q_VALVE_3" )
      Move(in := "DB_Webserver".Act_Weight_3, out1 => "DB_Webserver".sql_Weight3_Setting)
   END_RUNG
   RUNG wire#w1
      Contact( "Q_DC_TRON" )
      Move(in := "DB_Webserver".Act_Time_Tron, out1 => "DB_Webserver".sql_Time_Tron_Setting)
   END_RUNG
   RUNG wire#w1
      Move(in := "DB_Webserver".Act_Weight_1, out1 => "DB_Webserver".sql_Weight1_Actual)
      Move(in := "DB_Webserver".Act_Weight_2, out1 => "DB_Webserver".sql_Weight2_Actual)
      Move(in := "DB_Webserver".Act_Weight_3, out1 => "DB_Webserver".sql_Weight3_Actual)
      Move(in := "DB_Webserver".Act_Time_Tron, out1 => "DB_Webserver".sql_Time_Tron_Actual)
   END_RUNG
   // the same network as SCL:
   IF "DB_Webserver".sql_insert_Trigger AND "Q_VALVE_1" THEN
       "DB_Webserver".sql_Weight1_Setting := "DB_Webserver".Act_Weight_1;
   END_IF;
   IF "DB_Webserver".sql_insert_Trigger AND "Q_VALVE_2" THEN
       "DB_Webserver".sql_Weight2_Setting := "DB_Webserver".Act_Weight_2;
   END_IF;
   IF "DB_Webserver".sql_insert_Trigger AND "Q_VALVE_3" THEN
       "DB_Webserver".sql_Weight3_Setting := "DB_Webserver".Act_Weight_3;
   END_IF;
   IF "DB_Webserver".sql_insert_Trigger AND "Q_DC_TRON" THEN
       "DB_Webserver".sql_Time_Tron_Setting := "DB_Webserver".Act_Time_Tron;
   END_IF;
   IF "DB_Webserver".sql_insert_Trigger THEN
       "DB_Webserver".sql_Weight1_Actual := "DB_Webserver".Act_Weight_1;
       "DB_Webserver".sql_Weight2_Actual := "DB_Webserver".Act_Weight_2;
       "DB_Webserver".sql_Weight3_Actual := "DB_Webserver".Act_Weight_3;
       "DB_Webserver".sql_Time_Tron_Actual := "DB_Webserver".Act_Time_Tron;
   END_IF;
END_REGION

REGION Network 12: Bit xóa dữ liệu SQL
   "TImer_SQL_Delete".TON(IN := "DB_Webserver".sql_delete_Trigger, PT := T#1s);
   IF "TImer_SQL_Delete".Q THEN "DB_Webserver".sql_delete_Trigger := FALSE; END_IF;
END_REGION

REGION Network 13: Cảm biến bồn trộn
   "TIMER_SIMU".TON(IN := NOT "AlwaysFALSE" AND "Q_DC_Export", PT := T#8s);
   IF "TIMER_SIMU".Q THEN "DB_Webserver".CB_Can := TRUE; END_IF;
   IF NOT "AlwaysFALSE" AND "Q_VALVE_1" THEN "DB_Webserver".CB_Can := FALSE; END_IF;
END_REGION
END_FUNCTION

FUNCTION "FC_AUTO_MODE" : Void   // FC2, LAD
{ S7_Optimized_Access := 'TRUE' }
VERSION : 0.1
   VAR_TEMP   // added for the SCL form of the ladder/FBD networks
      _w1 : Bool;
      _w2 : Bool;
      _w3 : Bool;
      _w4 : Bool;
      _w5 : Bool;
      _w6 : Bool;
   END_VAR
BEGIN

REGION Network 1: mô phỏng tăng trọng lượng
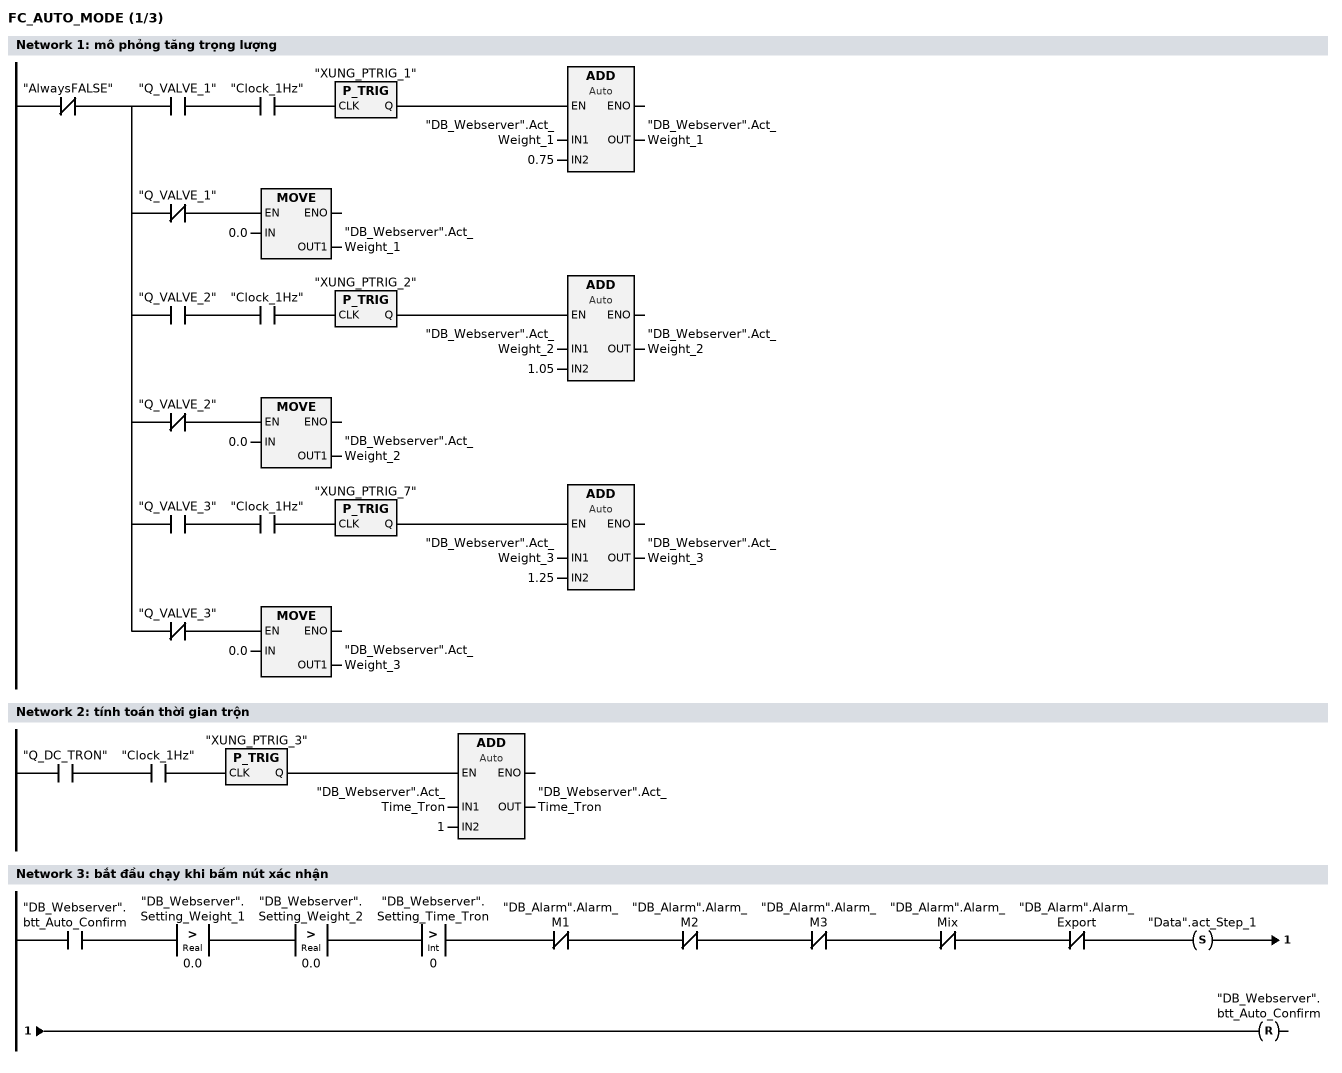
   RUNG wire#powerrail
      I_Contact( "AlwaysFALSE" )
      wire#w1
      Contact( "Q_VALVE_1" )
      Contact( "Clock_1Hz" )
      P_Trig( "XUNG_PTRIG_1" )
      Add(in1 := "DB_Webserver".Act_Weight_1, in2 := 0.75, out => "DB_Webserver".Act_Weight_1)
   END_RUNG
   RUNG wire#w1
      I_Contact( "Q_VALVE_1" )
      Move(in := 0.0, out1 => "DB_Webserver".Act_Weight_1)
   END_RUNG
   RUNG wire#w1
      Contact( "Q_VALVE_2" )
      Contact( "Clock_1Hz" )
      P_Trig( "XUNG_PTRIG_2" )
      Add(in1 := "DB_Webserver".Act_Weight_2, in2 := 1.05, out => "DB_Webserver".Act_Weight_2)
   END_RUNG
   RUNG wire#w1
      I_Contact( "Q_VALVE_2" )
      Move(in := 0.0, out1 => "DB_Webserver".Act_Weight_2)
   END_RUNG
   RUNG wire#w1
      Contact( "Q_VALVE_3" )
      Contact( "Clock_1Hz" )
      P_Trig( "XUNG_PTRIG_7" )
      Add(in1 := "DB_Webserver".Act_Weight_3, in2 := 1.25, out => "DB_Webserver".Act_Weight_3)
   END_RUNG
   RUNG wire#w1
      I_Contact( "Q_VALVE_3" )
      Move(in := 0.0, out1 => "DB_Webserver".Act_Weight_3)
   END_RUNG
   // the same network as SCL:
   #_w1 := NOT "AlwaysFALSE" AND "Q_VALVE_1" AND "Clock_1Hz";
   #_w2 := #_w1 AND NOT "XUNG_PTRIG_1";   // rising edge
   "XUNG_PTRIG_1" := #_w1;
   IF #_w2 THEN "DB_Webserver".Act_Weight_1 := "DB_Webserver".Act_Weight_1 + 0.75; END_IF;
   IF NOT "AlwaysFALSE" AND NOT "Q_VALVE_1" THEN "DB_Webserver".Act_Weight_1 := 0.0; END_IF;
   #_w3 := NOT "AlwaysFALSE" AND "Q_VALVE_2" AND "Clock_1Hz";
   #_w4 := #_w3 AND NOT "XUNG_PTRIG_2";   // rising edge
   "XUNG_PTRIG_2" := #_w3;
   IF #_w4 THEN "DB_Webserver".Act_Weight_2 := "DB_Webserver".Act_Weight_2 + 1.05; END_IF;
   IF NOT "AlwaysFALSE" AND NOT "Q_VALVE_2" THEN "DB_Webserver".Act_Weight_2 := 0.0; END_IF;
   #_w5 := NOT "AlwaysFALSE" AND "Q_VALVE_3" AND "Clock_1Hz";
   #_w6 := #_w5 AND NOT "XUNG_PTRIG_7";   // rising edge
   "XUNG_PTRIG_7" := #_w5;
   IF #_w6 THEN "DB_Webserver".Act_Weight_3 := "DB_Webserver".Act_Weight_3 + 1.25; END_IF;
   IF NOT "AlwaysFALSE" AND NOT "Q_VALVE_3" THEN "DB_Webserver".Act_Weight_3 := 0.0; END_IF;
END_REGION

REGION Network 2: tính toán thời gian trộn
   RUNG wire#powerrail
      Contact( "Q_DC_TRON" )
      Contact( "Clock_1Hz" )
      P_Trig( "XUNG_PTRIG_3" )
      Add(in1 := "DB_Webserver".Act_Time_Tron, in2 := 1, out => "DB_Webserver".Act_Time_Tron)
   END_RUNG
   // the same network as SCL:
   #_w1 := "Q_DC_TRON" AND "Clock_1Hz";
   #_w2 := #_w1 AND NOT "XUNG_PTRIG_3";   // rising edge
   "XUNG_PTRIG_3" := #_w1;
   IF #_w2 THEN "DB_Webserver".Act_Time_Tron := "DB_Webserver".Act_Time_Tron + 1; END_IF;
END_REGION

REGION Network 3: bắt đầu chạy khi bấm nút xác nhận
   RUNG wire#powerrail
      Contact( "DB_Webserver".btt_Auto_Confirm )
      { S7_Templates := "SrcType := Real" } GT_Contact(in1 := "DB_Webserver".Setting_Weight_1, in2 := 0.0)
      { S7_Templates := "SrcType := Real" } GT_Contact(in1 := "DB_Webserver".Setting_Weight_2, in2 := 0.0)
      { S7_Templates := "SrcType := Int" } GT_Contact(in1 := "DB_Webserver".Setting_Time_Tron, in2 := 0)
      I_Contact( "DB_Alarm".Alarm_M1 )
      I_Contact( "DB_Alarm".Alarm_M2 )
      I_Contact( "DB_Alarm".Alarm_M3 )
      I_Contact( "DB_Alarm".Alarm_Mix )
      I_Contact( "DB_Alarm".Alarm_Export )
      S_Coil( "Data".act_Step_1 )
      R_Coil( "DB_Webserver".btt_Auto_Confirm )
   END_RUNG
   // the same network as SCL:
   IF "DB_Webserver".btt_Auto_Confirm AND ("DB_Webserver".Setting_Weight_1 > 0.0) AND ("DB_Webserver".Setting_Weight_2 > 0.0) AND ("DB_Webserver".Setting_Time_Tron > 0) AND NOT "DB_Alarm".Alarm_M1 AND NOT "DB_Alarm".Alarm_M2 AND NOT "DB_Alarm".Alarm_M3 AND NOT "DB_Alarm".Alarm_Mix AND NOT "DB_Alarm".Alarm_Export THEN
       "Data".act_Step_1 := TRUE;
       "DB_Webserver".btt_Auto_Confirm := FALSE;
   END_IF;
END_REGION

REGION Network 4: Giai đoạn 1
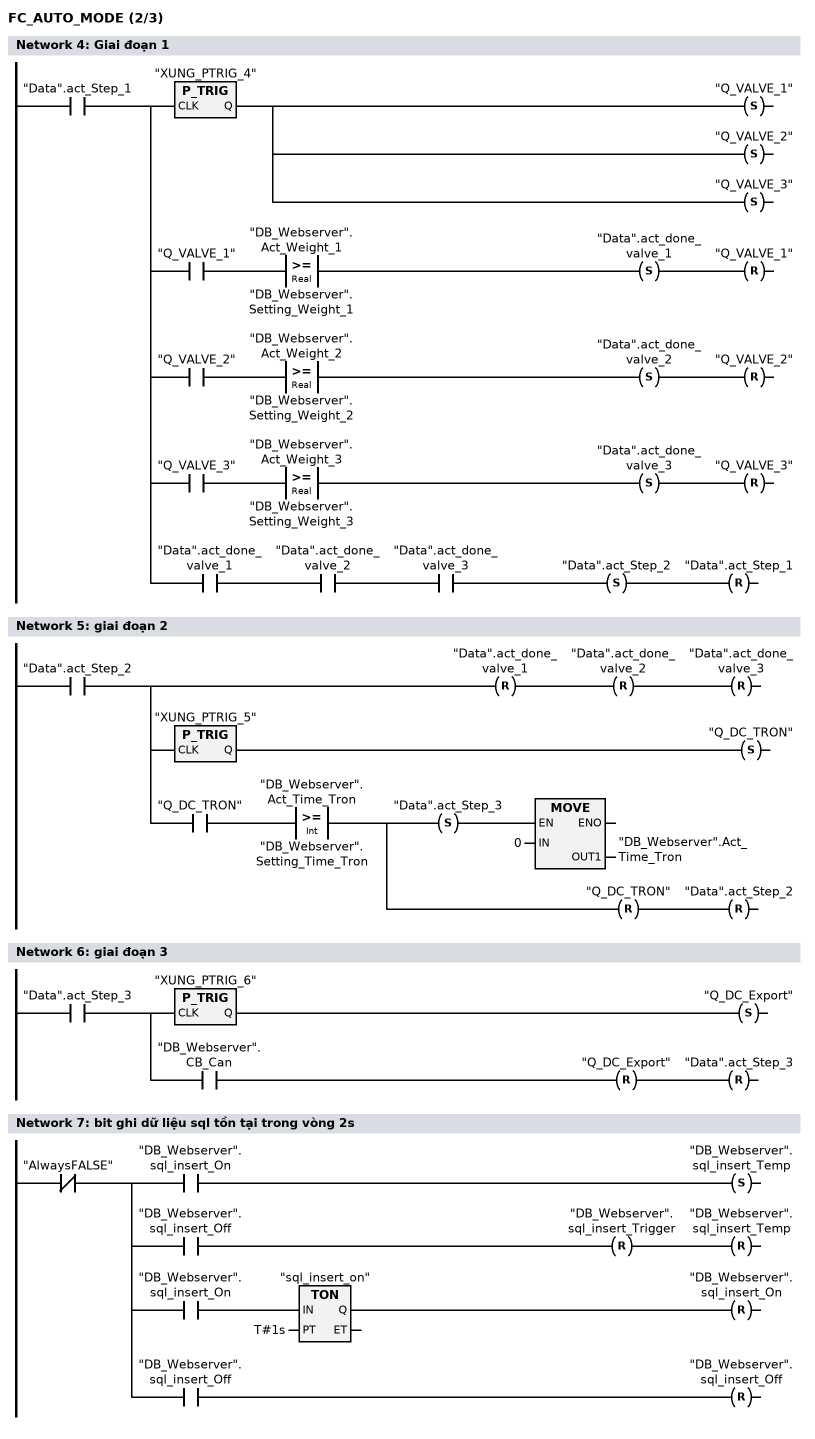
   RUNG wire#powerrail
      Contact( "Data".act_Step_1 )
      wire#w1
      P_Trig( "XUNG_PTRIG_4" )
      wire#w2
      S_Coil( "Q_VALVE_1" )
   END_RUNG
   RUNG wire#w2
      S_Coil( "Q_VALVE_2" )
   END_RUNG
   RUNG wire#w2
      S_Coil( "Q_VALVE_3" )
   END_RUNG
   RUNG wire#w1
      Contact( "Q_VALVE_1" )
      { S7_Templates := "SrcType := Real" } GE_Contact(in1 := "DB_Webserver".Act_Weight_1, in2 := "DB_Webserver".Setting_Weight_1)
      S_Coil( "Data".act_done_valve_1 )
      R_Coil( "Q_VALVE_1" )
   END_RUNG
   RUNG wire#w1
      Contact( "Q_VALVE_2" )
      { S7_Templates := "SrcType := Real" } GE_Contact(in1 := "DB_Webserver".Act_Weight_2, in2 := "DB_Webserver".Setting_Weight_2)
      S_Coil( "Data".act_done_valve_2 )
      R_Coil( "Q_VALVE_2" )
   END_RUNG
   RUNG wire#w1
      Contact( "Q_VALVE_3" )
      { S7_Templates := "SrcType := Real" } GE_Contact(in1 := "DB_Webserver".Act_Weight_3, in2 := "DB_Webserver".Setting_Weight_3)
      S_Coil( "Data".act_done_valve_3 )
      R_Coil( "Q_VALVE_3" )
   END_RUNG
   RUNG wire#w1
      Contact( "Data".act_done_valve_1 )
      Contact( "Data".act_done_valve_2 )
      Contact( "Data".act_done_valve_3 )
      S_Coil( "Data".act_Step_2 )
      R_Coil( "Data".act_Step_1 )
   END_RUNG
   // the same network as SCL:
   #_w1 := "Data".act_Step_1 AND NOT "XUNG_PTRIG_4";   // rising edge
   "XUNG_PTRIG_4" := "Data".act_Step_1;
   IF #_w1 THEN
       "Q_VALVE_1" := TRUE;
       "Q_VALVE_2" := TRUE;
       "Q_VALVE_3" := TRUE;
   END_IF;
   IF "Data".act_Step_1 AND "Q_VALVE_1" AND ("DB_Webserver".Act_Weight_1 >= "DB_Webserver".Setting_Weight_1) THEN
       "Data".act_done_valve_1 := TRUE;
       "Q_VALVE_1" := FALSE;
   END_IF;
   IF "Data".act_Step_1 AND "Q_VALVE_2" AND ("DB_Webserver".Act_Weight_2 >= "DB_Webserver".Setting_Weight_2) THEN
       "Data".act_done_valve_2 := TRUE;
       "Q_VALVE_2" := FALSE;
   END_IF;
   IF "Data".act_Step_1 AND "Q_VALVE_3" AND ("DB_Webserver".Act_Weight_3 >= "DB_Webserver".Setting_Weight_3) THEN
       "Data".act_done_valve_3 := TRUE;
       "Q_VALVE_3" := FALSE;
   END_IF;
   IF "Data".act_Step_1 AND "Data".act_done_valve_1 AND "Data".act_done_valve_2 AND "Data".act_done_valve_3 THEN
       "Data".act_Step_2 := TRUE;
       "Data".act_Step_1 := FALSE;
   END_IF;
END_REGION

REGION Network 5: giai đoạn 2
   RUNG wire#powerrail
      Contact( "Data".act_Step_2 )
      wire#w1
      R_Coil( "Data".act_done_valve_1 )
      R_Coil( "Data".act_done_valve_2 )
      R_Coil( "Data".act_done_valve_3 )
   END_RUNG
   RUNG wire#w1
      P_Trig( "XUNG_PTRIG_5" )
      S_Coil( "Q_DC_TRON" )
   END_RUNG
   RUNG wire#w1
      Contact( "Q_DC_TRON" )
      { S7_Templates := "SrcType := Int" } GE_Contact(in1 := "DB_Webserver".Act_Time_Tron, in2 := "DB_Webserver".Setting_Time_Tron)
      wire#w2
      S_Coil( "Data".act_Step_3 )
      Move(in := 0, out1 => "DB_Webserver".Act_Time_Tron)
   END_RUNG
   RUNG wire#w2
      R_Coil( "Q_DC_TRON" )
      R_Coil( "Data".act_Step_2 )
   END_RUNG
   // the same network as SCL:
   IF "Data".act_Step_2 THEN
       "Data".act_done_valve_1 := FALSE;
       "Data".act_done_valve_2 := FALSE;
       "Data".act_done_valve_3 := FALSE;
   END_IF;
   #_w1 := "Data".act_Step_2 AND NOT "XUNG_PTRIG_5";   // rising edge
   "XUNG_PTRIG_5" := "Data".act_Step_2;
   IF #_w1 THEN "Q_DC_TRON" := TRUE; END_IF;
   IF "Data".act_Step_2 AND "Q_DC_TRON" AND ("DB_Webserver".Act_Time_Tron >= "DB_Webserver".Setting_Time_Tron) THEN
       "Data".act_Step_3 := TRUE;
   END_IF;
   #_w2 := "Data".act_Step_2 AND "Q_DC_TRON" AND ("DB_Webserver".Act_Time_Tron >= "DB_Webserver".Setting_Time_Tron);
   IF #_w2 THEN
       "DB_Webserver".Act_Time_Tron := 0;
       "Q_DC_TRON" := FALSE;
       "Data".act_Step_2 := FALSE;
   END_IF;
END_REGION

REGION Network 6: giai đoạn 3
   RUNG wire#powerrail
      Contact( "Data".act_Step_3 )
      wire#w1
      P_Trig( "XUNG_PTRIG_6" )
      S_Coil( "Q_DC_Export" )
   END_RUNG
   RUNG wire#w1
      Contact( "DB_Webserver".CB_Can )
      R_Coil( "Q_DC_Export" )
      R_Coil( "Data".act_Step_3 )
   END_RUNG
   // the same network as SCL:
   #_w1 := "Data".act_Step_3 AND NOT "XUNG_PTRIG_6";   // rising edge
   "XUNG_PTRIG_6" := "Data".act_Step_3;
   IF #_w1 THEN "Q_DC_Export" := TRUE; END_IF;
   IF "Data".act_Step_3 AND "DB_Webserver".CB_Can THEN
       "Q_DC_Export" := FALSE;
       "Data".act_Step_3 := FALSE;
   END_IF;
END_REGION

REGION Network 7: bit ghi dữ liệu sql tồn tại trong vòng 2s
   IF NOT "AlwaysFALSE" AND "DB_Webserver".sql_insert_On THEN "DB_Webserver".sql_insert_Temp := TRUE; END_IF;
   IF NOT "AlwaysFALSE" AND "DB_Webserver".sql_insert_Off THEN
       "DB_Webserver".sql_insert_Trigger := FALSE;
       "DB_Webserver".sql_insert_Temp := FALSE;
   END_IF;
   "sql_insert_on".TON(IN := NOT "AlwaysFALSE" AND "DB_Webserver".sql_insert_On, PT := T#1s);
   IF "sql_insert_on".Q THEN "DB_Webserver".sql_insert_On := FALSE; END_IF;
   IF NOT "AlwaysFALSE" AND "DB_Webserver".sql_insert_Off THEN
       "DB_Webserver".sql_insert_Off := FALSE;
   END_IF;
END_REGION

REGION Network 8: bit ghi dữ liệu sql tồn tại trong vòng 2s
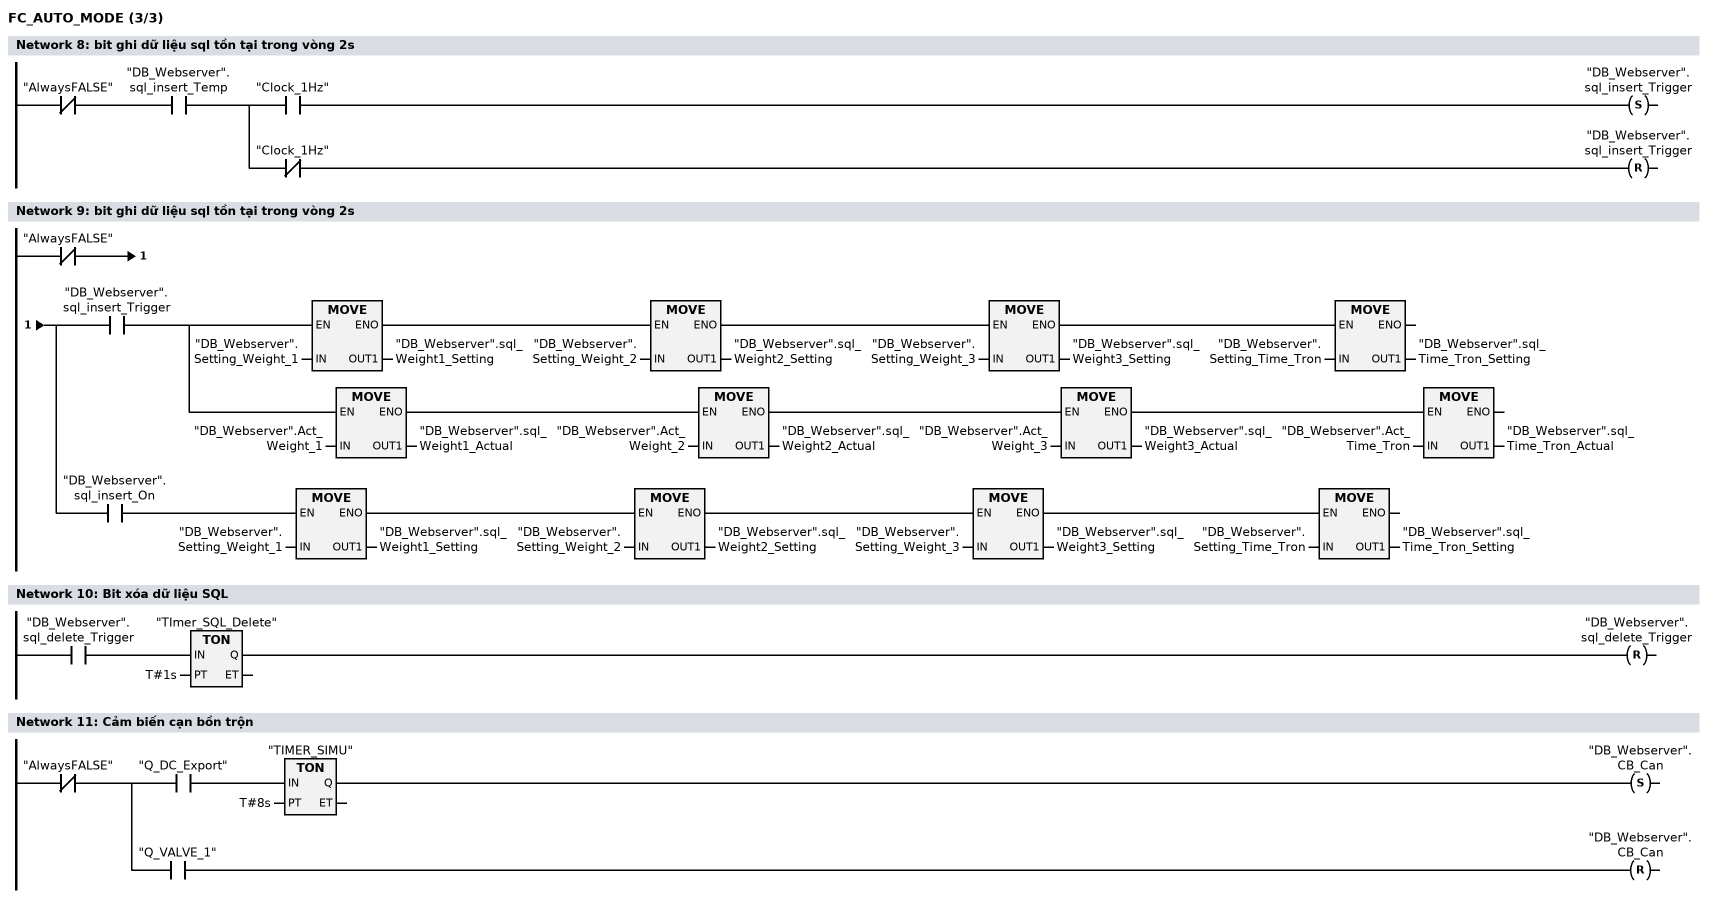
   RUNG wire#powerrail
      I_Contact( "AlwaysFALSE" )
      Contact( "DB_Webserver".sql_insert_Temp )
      wire#w1
      Contact( "Clock_1Hz" )
      S_Coil( "DB_Webserver".sql_insert_Trigger )
   END_RUNG
   RUNG wire#w1
      I_Contact( "Clock_1Hz" )
      R_Coil( "DB_Webserver".sql_insert_Trigger )
   END_RUNG
   // the same network as SCL:
   #_w1 := NOT "AlwaysFALSE" AND "DB_Webserver".sql_insert_Temp;
   IF #_w1 AND "Clock_1Hz" THEN "DB_Webserver".sql_insert_Trigger := TRUE; END_IF;
   IF #_w1 AND NOT "Clock_1Hz" THEN "DB_Webserver".sql_insert_Trigger := FALSE; END_IF;
END_REGION

REGION Network 9: bit ghi dữ liệu sql tồn tại trong vòng 2s
   RUNG wire#powerrail
      I_Contact( "AlwaysFALSE" )
      wire#w1
      Contact( "DB_Webserver".sql_insert_Trigger )
      wire#w2
      Move(in := "DB_Webserver".Setting_Weight_1, out1 => "DB_Webserver".sql_Weight1_Setting)
      Move(in := "DB_Webserver".Setting_Weight_2, out1 => "DB_Webserver".sql_Weight2_Setting)
      Move(in := "DB_Webserver".Setting_Weight_3, out1 => "DB_Webserver".sql_Weight3_Setting)
      Move(in := "DB_Webserver".Setting_Time_Tron, out1 => "DB_Webserver".sql_Time_Tron_Setting)
   END_RUNG
   RUNG wire#w2
      Move(in := "DB_Webserver".Act_Weight_1, out1 => "DB_Webserver".sql_Weight1_Actual)
      Move(in := "DB_Webserver".Act_Weight_2, out1 => "DB_Webserver".sql_Weight2_Actual)
      Move(in := "DB_Webserver".Act_Weight_3, out1 => "DB_Webserver".sql_Weight3_Actual)
      Move(in := "DB_Webserver".Act_Time_Tron, out1 => "DB_Webserver".sql_Time_Tron_Actual)
   END_RUNG
   RUNG wire#w1
      Contact( "DB_Webserver".sql_insert_On )
      Move(in := "DB_Webserver".Setting_Weight_1, out1 => "DB_Webserver".sql_Weight1_Setting)
      Move(in := "DB_Webserver".Setting_Weight_2, out1 => "DB_Webserver".sql_Weight2_Setting)
      Move(in := "DB_Webserver".Setting_Weight_3, out1 => "DB_Webserver".sql_Weight3_Setting)
      Move(in := "DB_Webserver".Setting_Time_Tron, out1 => "DB_Webserver".sql_Time_Tron_Setting)
   END_RUNG
   // the same network as SCL:
   IF NOT "AlwaysFALSE" AND "DB_Webserver".sql_insert_Trigger THEN
       "DB_Webserver".sql_Weight1_Setting := "DB_Webserver".Setting_Weight_1;
       "DB_Webserver".sql_Weight2_Setting := "DB_Webserver".Setting_Weight_2;
       "DB_Webserver".sql_Weight3_Setting := "DB_Webserver".Setting_Weight_3;
       "DB_Webserver".sql_Time_Tron_Setting := "DB_Webserver".Setting_Time_Tron;
       "DB_Webserver".sql_Weight1_Actual := "DB_Webserver".Act_Weight_1;
       "DB_Webserver".sql_Weight2_Actual := "DB_Webserver".Act_Weight_2;
       "DB_Webserver".sql_Weight3_Actual := "DB_Webserver".Act_Weight_3;
       "DB_Webserver".sql_Time_Tron_Actual := "DB_Webserver".Act_Time_Tron;
   END_IF;
   IF NOT "AlwaysFALSE" AND "DB_Webserver".sql_insert_On THEN
       "DB_Webserver".sql_Weight1_Setting := "DB_Webserver".Setting_Weight_1;
       "DB_Webserver".sql_Weight2_Setting := "DB_Webserver".Setting_Weight_2;
       "DB_Webserver".sql_Weight3_Setting := "DB_Webserver".Setting_Weight_3;
       "DB_Webserver".sql_Time_Tron_Setting := "DB_Webserver".Setting_Time_Tron;
   END_IF;
END_REGION

REGION Network 10: Bit xóa dữ liệu SQL
   "TImer_SQL_Delete".TON(IN := "DB_Webserver".sql_delete_Trigger, PT := T#1s);
   IF "TImer_SQL_Delete".Q THEN "DB_Webserver".sql_delete_Trigger := FALSE; END_IF;
END_REGION

REGION Network 11: Cảm biến cạn bồn trộn
   "TIMER_SIMU".TON(IN := NOT "AlwaysFALSE" AND "Q_DC_Export", PT := T#8s);
   IF "TIMER_SIMU".Q THEN "DB_Webserver".CB_Can := TRUE; END_IF;
   IF NOT "AlwaysFALSE" AND "Q_VALVE_1" THEN "DB_Webserver".CB_Can := FALSE; END_IF;
END_REGION
END_FUNCTION

FUNCTION "FC_EQUIPMENT_STATUS" : Void   // FC3, LAD
{ S7_Optimized_Access := 'TRUE' }
VERSION : 0.1
   VAR_TEMP   // added for the SCL form of the ladder/FBD networks
      _w1 : Bool;
   END_VAR
BEGIN

REGION Network 1: hiển thị trạng thái đèn
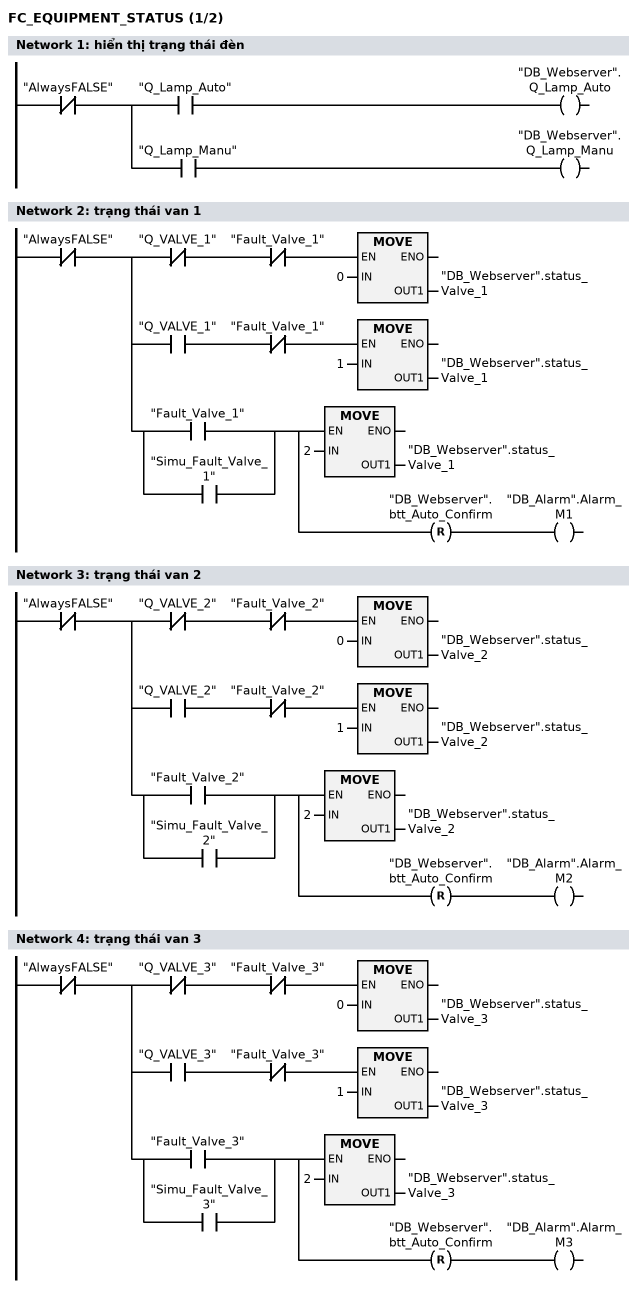
   RUNG wire#powerrail
      I_Contact( "AlwaysFALSE" )
      wire#w1
      Contact( "Q_Lamp_Auto" )
      Coil( "DB_Webserver".Q_Lamp_Auto )
   END_RUNG
   RUNG wire#w1
      Contact( "Q_Lamp_Manu" )
      Coil( "DB_Webserver".Q_Lamp_Manu )
   END_RUNG
   // the same network as SCL:
   "DB_Webserver".Q_Lamp_Auto := NOT "AlwaysFALSE" AND "Q_Lamp_Auto";
   "DB_Webserver".Q_Lamp_Manu := NOT "AlwaysFALSE" AND "Q_Lamp_Manu";
END_REGION

REGION Network 2: trạng thái van 1
   RUNG wire#powerrail
      I_Contact( "AlwaysFALSE" )
      wire#w1
      I_Contact( "Q_VALVE_1" )
      I_Contact( "Fault_Valve_1" )
      Move(in := 0, out1 => "DB_Webserver".status_Valve_1)
   END_RUNG
   RUNG wire#w1
      Contact( "Q_VALVE_1" )
      I_Contact( "Fault_Valve_1" )
      Move(in := 1, out1 => "DB_Webserver".status_Valve_1)
   END_RUNG
   RUNG wire#w1
      Contact( "Fault_Valve_1" )
      wire#w2
      Move(in := 2, out1 => "DB_Webserver".status_Valve_1)
   END_RUNG
   RUNG wire#w1
      Contact( "Simu_Fault_Valve_1" )
   END_RUNG wire#w2
   RUNG wire#w2
      R_Coil( "DB_Webserver".btt_Auto_Confirm )
      Coil( "DB_Alarm".Alarm_M1 )
   END_RUNG
   // the same network as SCL:
   IF NOT "AlwaysFALSE" AND NOT "Q_VALVE_1" AND NOT "Fault_Valve_1" THEN
       "DB_Webserver".status_Valve_1 := 0;
   END_IF;
   IF NOT "AlwaysFALSE" AND "Q_VALVE_1" AND NOT "Fault_Valve_1" THEN
       "DB_Webserver".status_Valve_1 := 1;
   END_IF;
   #_w1 := NOT "AlwaysFALSE" AND ("Fault_Valve_1" OR "Simu_Fault_Valve_1");
   IF #_w1 THEN
       "DB_Webserver".status_Valve_1 := 2;
       "DB_Webserver".btt_Auto_Confirm := FALSE;
   END_IF;
   "DB_Alarm".Alarm_M1 := #_w1;
END_REGION

REGION Network 3: trạng thái van 2
   RUNG wire#powerrail
      I_Contact( "AlwaysFALSE" )
      wire#w1
      I_Contact( "Q_VALVE_2" )
      I_Contact( "Fault_Valve_2" )
      Move(in := 0, out1 => "DB_Webserver".status_Valve_2)
   END_RUNG
   RUNG wire#w1
      Contact( "Q_VALVE_2" )
      I_Contact( "Fault_Valve_2" )
      Move(in := 1, out1 => "DB_Webserver".status_Valve_2)
   END_RUNG
   RUNG wire#w1
      Contact( "Fault_Valve_2" )
      wire#w2
      Move(in := 2, out1 => "DB_Webserver".status_Valve_2)
   END_RUNG
   RUNG wire#w1
      Contact( "Simu_Fault_Valve_2" )
   END_RUNG wire#w2
   RUNG wire#w2
      R_Coil( "DB_Webserver".btt_Auto_Confirm )
      Coil( "DB_Alarm".Alarm_M2 )
   END_RUNG
   // the same network as SCL:
   IF NOT "AlwaysFALSE" AND NOT "Q_VALVE_2" AND NOT "Fault_Valve_2" THEN
       "DB_Webserver".status_Valve_2 := 0;
   END_IF;
   IF NOT "AlwaysFALSE" AND "Q_VALVE_2" AND NOT "Fault_Valve_2" THEN
       "DB_Webserver".status_Valve_2 := 1;
   END_IF;
   #_w1 := NOT "AlwaysFALSE" AND ("Fault_Valve_2" OR "Simu_Fault_Valve_2");
   IF #_w1 THEN
       "DB_Webserver".status_Valve_2 := 2;
       "DB_Webserver".btt_Auto_Confirm := FALSE;
   END_IF;
   "DB_Alarm".Alarm_M2 := #_w1;
END_REGION

REGION Network 4: trạng thái van 3
   RUNG wire#powerrail
      I_Contact( "AlwaysFALSE" )
      wire#w1
      I_Contact( "Q_VALVE_3" )
      I_Contact( "Fault_Valve_3" )
      Move(in := 0, out1 => "DB_Webserver".status_Valve_3)
   END_RUNG
   RUNG wire#w1
      Contact( "Q_VALVE_3" )
      I_Contact( "Fault_Valve_3" )
      Move(in := 1, out1 => "DB_Webserver".status_Valve_3)
   END_RUNG
   RUNG wire#w1
      Contact( "Fault_Valve_3" )
      wire#w2
      Move(in := 2, out1 => "DB_Webserver".status_Valve_3)
   END_RUNG
   RUNG wire#w1
      Contact( "Simu_Fault_Valve_3" )
   END_RUNG wire#w2
   RUNG wire#w2
      R_Coil( "DB_Webserver".btt_Auto_Confirm )
      Coil( "DB_Alarm".Alarm_M3 )
   END_RUNG
   // the same network as SCL:
   IF NOT "AlwaysFALSE" AND NOT "Q_VALVE_3" AND NOT "Fault_Valve_3" THEN
       "DB_Webserver".status_Valve_3 := 0;
   END_IF;
   IF NOT "AlwaysFALSE" AND "Q_VALVE_3" AND NOT "Fault_Valve_3" THEN
       "DB_Webserver".status_Valve_3 := 1;
   END_IF;
   #_w1 := NOT "AlwaysFALSE" AND ("Fault_Valve_3" OR "Simu_Fault_Valve_3");
   IF #_w1 THEN
       "DB_Webserver".status_Valve_3 := 2;
       "DB_Webserver".btt_Auto_Confirm := FALSE;
   END_IF;
   "DB_Alarm".Alarm_M3 := #_w1;
END_REGION

REGION Network 5: trạng thái động cơ
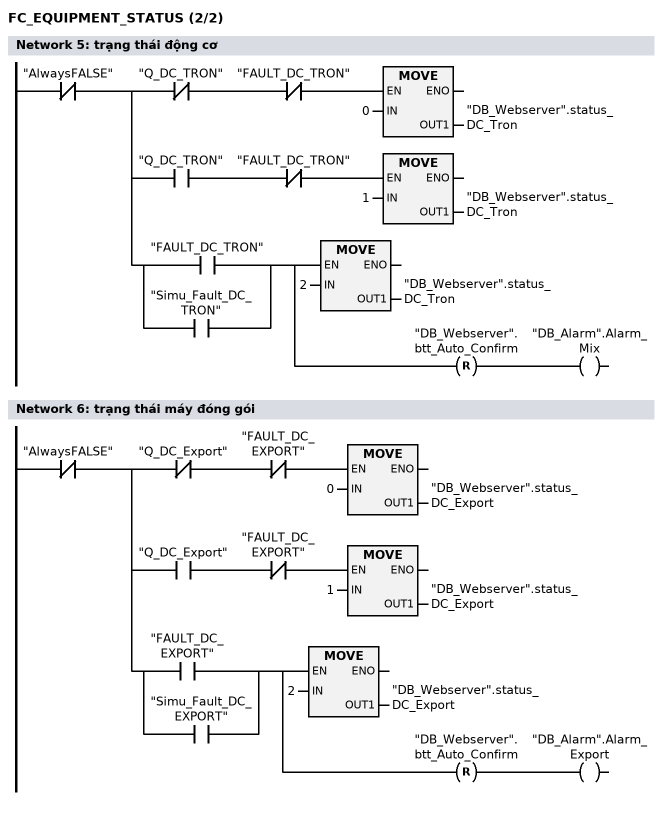
   RUNG wire#powerrail
      I_Contact( "AlwaysFALSE" )
      wire#w1
      I_Contact( "Q_DC_TRON" )
      I_Contact( "FAULT_DC_TRON" )
      Move(in := 0, out1 => "DB_Webserver".status_DC_Tron)
   END_RUNG
   RUNG wire#w1
      Contact( "Q_DC_TRON" )
      I_Contact( "FAULT_DC_TRON" )
      Move(in := 1, out1 => "DB_Webserver".status_DC_Tron)
   END_RUNG
   RUNG wire#w1
      Contact( "FAULT_DC_TRON" )
      wire#w2
      Move(in := 2, out1 => "DB_Webserver".status_DC_Tron)
   END_RUNG
   RUNG wire#w1
      Contact( "Simu_Fault_DC_TRON" )
   END_RUNG wire#w2
   RUNG wire#w2
      R_Coil( "DB_Webserver".btt_Auto_Confirm )
      Coil( "DB_Alarm".Alarm_Mix )
   END_RUNG
   // the same network as SCL:
   IF NOT "AlwaysFALSE" AND NOT "Q_DC_TRON" AND NOT "FAULT_DC_TRON" THEN
       "DB_Webserver".status_DC_Tron := 0;
   END_IF;
   IF NOT "AlwaysFALSE" AND "Q_DC_TRON" AND NOT "FAULT_DC_TRON" THEN
       "DB_Webserver".status_DC_Tron := 1;
   END_IF;
   #_w1 := NOT "AlwaysFALSE" AND ("FAULT_DC_TRON" OR "Simu_Fault_DC_TRON");
   IF #_w1 THEN
       "DB_Webserver".status_DC_Tron := 2;
       "DB_Webserver".btt_Auto_Confirm := FALSE;
   END_IF;
   "DB_Alarm".Alarm_Mix := #_w1;
END_REGION

REGION Network 6: trạng thái máy đóng gói
   RUNG wire#powerrail
      I_Contact( "AlwaysFALSE" )
      wire#w1
      I_Contact( "Q_DC_Export" )
      I_Contact( "FAULT_DC_EXPORT" )
      Move(in := 0, out1 => "DB_Webserver".status_DC_Export)
   END_RUNG
   RUNG wire#w1
      Contact( "Q_DC_Export" )
      I_Contact( "FAULT_DC_EXPORT" )
      Move(in := 1, out1 => "DB_Webserver".status_DC_Export)
   END_RUNG
   RUNG wire#w1
      Contact( "FAULT_DC_EXPORT" )
      wire#w2
      Move(in := 2, out1 => "DB_Webserver".status_DC_Export)
   END_RUNG
   RUNG wire#w1
      Contact( "Simu_Fault_DC_EXPORT" )
   END_RUNG wire#w2
   RUNG wire#w2
      R_Coil( "DB_Webserver".btt_Auto_Confirm )
      Coil( "DB_Alarm".Alarm_Export )
   END_RUNG
   // the same network as SCL:
   IF NOT "AlwaysFALSE" AND NOT "Q_DC_Export" AND NOT "FAULT_DC_EXPORT" THEN
       "DB_Webserver".status_DC_Export := 0;
   END_IF;
   IF NOT "AlwaysFALSE" AND "Q_DC_Export" AND NOT "FAULT_DC_EXPORT" THEN
       "DB_Webserver".status_DC_Export := 1;
   END_IF;
   #_w1 := NOT "AlwaysFALSE" AND ("FAULT_DC_EXPORT" OR "Simu_Fault_DC_EXPORT");
   IF #_w1 THEN
       "DB_Webserver".status_DC_Export := 2;
       "DB_Webserver".btt_Auto_Confirm := FALSE;
   END_IF;
   "DB_Alarm".Alarm_Export := #_w1;
END_REGION
END_FUNCTION

ORGANIZATION_BLOCK "Main"   // OB1, LAD, ProgramCycle
TITLE = "Main Program Sweep (Cycle)"
{ S7_Optimized_Access := 'TRUE' }
VERSION : 0.1
   VAR_INPUT
      Initial_Call : Bool;   // Initial call of this OB
      Remanence : Bool;   // =True, if remanent data are available
   END_VAR
BEGIN

REGION Network 1: chế độ tự động
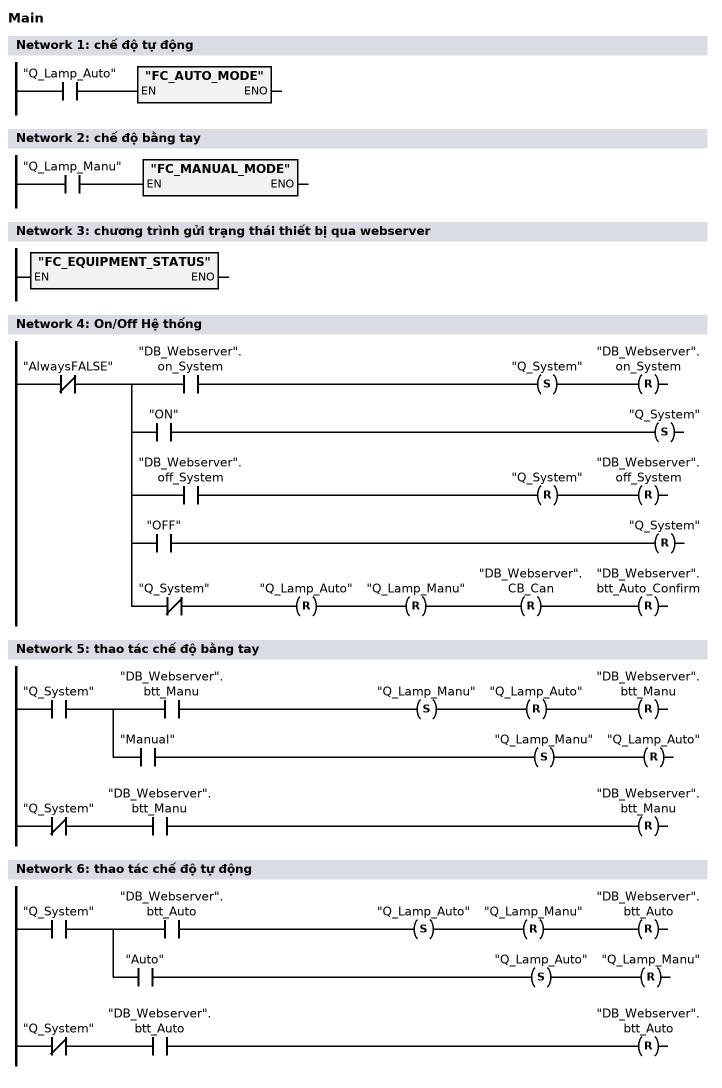
   RUNG wire#powerrail
      Contact( "Q_Lamp_Auto" )
      "FC_AUTO_MODE"()
   END_RUNG
   // the same network as SCL:
   IF "Q_Lamp_Auto" THEN "FC_AUTO_MODE"(); END_IF;
END_REGION

REGION Network 2: chế độ bằng tay
   RUNG wire#powerrail
      Contact( "Q_Lamp_Manu" )
      "FC_MANUAL_MODE"()
   END_RUNG
   // the same network as SCL:
   IF "Q_Lamp_Manu" THEN "FC_MANUAL_MODE"(); END_IF;
END_REGION

REGION Network 3: chương trình gửi trạng thái thiết bị qua webserver
   RUNG wire#powerrail
      "FC_EQUIPMENT_STATUS"()
   END_RUNG
   // the same network as SCL:
   "FC_EQUIPMENT_STATUS"();
END_REGION

REGION Network 4: On/Off Hệ thống
   RUNG wire#powerrail
      I_Contact( "AlwaysFALSE" )
      wire#w1
      Contact( "DB_Webserver".on_System )
      S_Coil( "Q_System" )
      R_Coil( "DB_Webserver".on_System )
   END_RUNG
   RUNG wire#w1
      Contact( "ON" )
      S_Coil( "Q_System" )
   END_RUNG
   RUNG wire#w1
      Contact( "DB_Webserver".off_System )
      R_Coil( "Q_System" )
      R_Coil( "DB_Webserver".off_System )
   END_RUNG
   RUNG wire#w1
      Contact( "OFF" )
      R_Coil( "Q_System" )
   END_RUNG
   RUNG wire#w1
      I_Contact( "Q_System" )
      R_Coil( "Q_Lamp_Auto" )
      R_Coil( "Q_Lamp_Manu" )
      R_Coil( "DB_Webserver".CB_Can )
      R_Coil( "DB_Webserver".btt_Auto_Confirm )
   END_RUNG
   // the same network as SCL:
   IF NOT "AlwaysFALSE" AND "DB_Webserver".on_System THEN
       "Q_System" := TRUE;
       "DB_Webserver".on_System := FALSE;
   END_IF;
   IF NOT "AlwaysFALSE" AND "ON" THEN "Q_System" := TRUE; END_IF;
   IF NOT "AlwaysFALSE" AND "DB_Webserver".off_System THEN
       "Q_System" := FALSE;
       "DB_Webserver".off_System := FALSE;
   END_IF;
   IF NOT "AlwaysFALSE" AND "OFF" THEN "Q_System" := FALSE; END_IF;
   IF NOT "AlwaysFALSE" AND NOT "Q_System" THEN
       "Q_Lamp_Auto" := FALSE;
       "Q_Lamp_Manu" := FALSE;
       "DB_Webserver".CB_Can := FALSE;
       "DB_Webserver".btt_Auto_Confirm := FALSE;
   END_IF;
END_REGION

REGION Network 5: thao tác chế độ bằng tay
   RUNG wire#powerrail
      Contact( "Q_System" )
      wire#w1
      Contact( "DB_Webserver".btt_Manu )
      S_Coil( "Q_Lamp_Manu" )
      R_Coil( "Q_Lamp_Auto" )
      R_Coil( "DB_Webserver".btt_Manu )
   END_RUNG
   RUNG wire#w1
      Contact( "Manual" )
      S_Coil( "Q_Lamp_Manu" )
      R_Coil( "Q_Lamp_Auto" )
   END_RUNG
   RUNG wire#powerrail
      I_Contact( "Q_System" )
      Contact( "DB_Webserver".btt_Manu )
      R_Coil( "DB_Webserver".btt_Manu )
   END_RUNG
   // the same network as SCL:
   IF "Q_System" AND "DB_Webserver".btt_Manu THEN
       "Q_Lamp_Manu" := TRUE;
       "Q_Lamp_Auto" := FALSE;
       "DB_Webserver".btt_Manu := FALSE;
   END_IF;
   IF "Q_System" AND "Manual" THEN
       "Q_Lamp_Manu" := TRUE;
       "Q_Lamp_Auto" := FALSE;
   END_IF;
   IF NOT "Q_System" AND "DB_Webserver".btt_Manu THEN "DB_Webserver".btt_Manu := FALSE; END_IF;
END_REGION

REGION Network 6: thao tác chế độ tự động
   RUNG wire#powerrail
      Contact( "Q_System" )
      wire#w1
      Contact( "DB_Webserver".btt_Auto )
      S_Coil( "Q_Lamp_Auto" )
      R_Coil( "Q_Lamp_Manu" )
      R_Coil( "DB_Webserver".btt_Auto )
   END_RUNG
   RUNG wire#w1
      Contact( "Auto" )
      S_Coil( "Q_Lamp_Auto" )
      R_Coil( "Q_Lamp_Manu" )
   END_RUNG
   RUNG wire#powerrail
      I_Contact( "Q_System" )
      Contact( "DB_Webserver".btt_Auto )
      R_Coil( "DB_Webserver".btt_Auto )
   END_RUNG
   // the same network as SCL:
   IF "Q_System" AND "DB_Webserver".btt_Auto THEN
       "Q_Lamp_Auto" := TRUE;
       "Q_Lamp_Manu" := FALSE;
       "DB_Webserver".btt_Auto := FALSE;
   END_IF;
   IF "Q_System" AND "Auto" THEN
       "Q_Lamp_Auto" := TRUE;
       "Q_Lamp_Manu" := FALSE;
   END_IF;
   IF NOT "Q_System" AND "DB_Webserver".btt_Auto THEN "DB_Webserver".btt_Auto := FALSE; END_IF;
END_REGION
END_ORGANIZATION_BLOCK